//     PlcTask Inputs/GLOBAL.mtcs.parts.cover.parts.io.parts.slot11.wcState <-> WcState/WcState
//     PlcTask Outputs/GLOBAL.mtcs.parts.cover.parts.bottom.parts.p3.parts.motorRelay.digitalOutput <-> Channel 1/Output
//     PlcTask Outputs/GLOBAL.mtcs.parts.cover.parts.bottom.parts.p4.parts.motorRelay.digitalOutput <-> Channel 2/Output
//   MTCS/MTCS Instance <-> ECAT (EtherCAT)/Pumps room star point - coupler (EK1101)/Pumps room star point - Slot 1 (EK1122)/REM star point (CU1128)/Cover coupler (EK1101)/Cover slot 12 (relays magnet top-bot, EL2622)
//     PlcTask Inputs/GLOBAL.mtcs.parts.cover.parts.io.parts.slot12.infoData <-> InfoData/State
//     PlcTask Inputs/GLOBAL.mtcs.parts.cover.parts.io.parts.slot12.wcState <-> WcState/WcState
//     PlcTask Outputs/GLOBAL.mtcs.parts.cover.parts.bottom.parts.magnetsRelay.digitalOutput <-> Channel 2/Output
//     PlcTask Outputs/GLOBAL.mtcs.parts.cover.parts.top.parts.magnetsRelay.digitalOutput <-> Channel 1/Output
//   MTCS/MTCS Instance <-> ECAT (EtherCAT)/Pumps room star point - coupler (EK1101)/Pumps room star point - Slot 1 (EK1122)/REM star point (CU1128)/Cover coupler (EK1101)/Cover slot 13 (multimeter, EL3681)
//     PlcTask Inputs/GLOBAL.mtcs.parts.cover.currentMeasurement.error <-> SAI Inputs/Error
//     PlcTask Inputs/GLOBAL.mtcs.parts.cover.currentMeasurement.microAmpsValue <-> SAI Inputs/Value
//     PlcTask Inputs/GLOBAL.mtcs.parts.cover.parts.io.parts.slot13.infoData <-> InfoData/State
//     PlcTask Inputs/GLOBAL.mtcs.parts.cover.parts.io.parts.slot13.wcState <-> WcState/WcState
//   MTCS/MTCS Instance <-> ECAT (EtherCAT)/Pumps room star point - coupler (EK1101)/Pumps room star point - Slot 1 (EK1122)/REM star point (CU1128)/Cover coupler (EK1101)/Cover slot 2 (analog out, EL4008)
//     PlcTask Inputs/GLOBAL.mtcs.parts.cover.parts.io.parts.slot2.infoData <-> InfoData/State
//     PlcTask Inputs/GLOBAL.mtcs.parts.cover.parts.io.parts.slot2.wcState <-> WcState/WcState
//   MTCS/MTCS Instance <-> ECAT (EtherCAT)/Pumps room star point - coupler (EK1101)/Pumps room star point - Slot 1 (EK1122)/REM star point (CU1128)/Cover coupler (EK1101)/Cover slot 3 (digital in, EL1088)
//     PlcTask Inputs/GLOBAL.mtcs.parts.cover.parts.bottom.parts.p{1..4}.encoderErrorSignal <-> Channel {5..8}/Input  (4 links)
//     PlcTask Inputs/GLOBAL.mtcs.parts.cover.parts.io.parts.slot3.infoData <-> InfoData/State
//     PlcTask Inputs/GLOBAL.mtcs.parts.cover.parts.io.parts.slot3.wcState <-> WcState/WcState
//     PlcTask Inputs/GLOBAL.mtcs.parts.cover.parts.top.parts.p{1..4}.encoderErrorSignal <-> Channel {1..4}/Input  (4 links)
//   MTCS/MTCS Instance <-> ECAT (EtherCAT)/Pumps room star point - coupler (EK1101)/Pumps room star point - Slot 1 (EK1122)/REM star point (CU1128)/Cover coupler (EK1101)/Cover slot 4 (enc top 1-2, EL5002)
//     PlcTask Inputs/GLOBAL.mtcs.parts.cover.parts.io.parts.slot4.infoData <-> InfoData/State
//     PlcTask Inputs/GLOBAL.mtcs.parts.cover.parts.io.parts.slot4.wcState <-> WcState/WcState
//   MTCS/MTCS Instance <-> ECAT (EtherCAT)/Pumps room star point - coupler (EK1101)/Pumps room star point - Slot 1 (EK1122)/REM star point (CU1128)/Cover coupler (EK1101)/Cover slot 5 (enc top 3-4, EL5002)
//     PlcTask Inputs/GLOBAL.mtcs.parts.cover.parts.io.parts.slot5.infoData <-> InfoData/State
//     PlcTask Inputs/GLOBAL.mtcs.parts.cover.parts.io.parts.slot5.wcState <-> WcState/WcState
//   MTCS/MTCS Instance <-> ECAT (EtherCAT)/Pumps room star point - coupler (EK1101)/Pumps room star point - Slot 1 (EK1122)/REM star point (CU1128)/Cover coupler (EK1101)/Cover slot 6 (enc bot 1-2, EL5002)
//     PlcTask Inputs/GLOBAL.mtcs.parts.cover.parts.io.parts.slot6.infoData <-> InfoData/State
//     PlcTask Inputs/GLOBAL.mtcs.parts.cover.parts.io.parts.slot6.wcState <-> WcState/WcState
//   MTCS/MTCS Instance <-> ECAT (EtherCAT)/Pumps room star point - coupler (EK1101)/Pumps room star point - Slot 1 (EK1122)/REM star point (CU1128)/Cover coupler (EK1101)/Cover slot 7 (enc bot 3-4, EL5002)
//     PlcTask Inputs/GLOBAL.mtcs.parts.cover.parts.io.parts.slot7.infoData <-> InfoData/State
//     PlcTask Inputs/GLOBAL.mtcs.parts.cover.parts.io.parts.slot7.wcState <-> WcState/WcState
//   MTCS/MTCS Instance <-> ECAT (EtherCAT)/Pumps room star point - coupler (EK1101)/Pumps room star point - Slot 1 (EK1122)/REM star point (CU1128)/Cover coupler (EK1101)/Cover slot 8 (relays top 1-2, EL2622)
//     PlcTask Inputs/GLOBAL.mtcs.parts.cover.parts.io.parts.slot8.infoData <-> InfoData/State
//     PlcTask Inputs/GLOBAL.mtcs.parts.cover.parts.io.parts.slot8.wcState <-> WcState/WcState
//     PlcTask Outputs/GLOBAL.mtcs.parts.cover.parts.top.parts.p1.parts.motorRelay.digitalOutput <-> Channel 1/Output
//     PlcTask Outputs/GLOBAL.mtcs.parts.cover.parts.top.parts.p2.parts.motorRelay.digitalOutput <-> Channel 2/Output
//   MTCS/MTCS Instance <-> ECAT (EtherCAT)/Pumps room star point - coupler (EK1101)/Pumps room star point - Slot 1 (EK1122)/REM star point (CU1128)/Cover coupler (EK1101)/Cover slot 9 (relays top 3-4, EL2622)
//     PlcTask Inputs/GLOBAL.mtcs.parts.cover.parts.io.parts.slot9.infoData <-> InfoData/State
//     PlcTask Inputs/GLOBAL.mtcs.parts.cover.parts.io.parts.slot9.wcState <-> WcState/WcState
//     PlcTask Outputs/GLOBAL.mtcs.parts.cover.parts.top.parts.p3.parts.motorRelay.digitalOutput <-> Channel 1/Output
//     PlcTask Outputs/GLOBAL.mtcs.parts.cover.parts.top.parts.p4.parts.motorRelay.digitalOutput <-> Channel 2/Output
//   MTCS/MTCS Instance <-> ECAT (EtherCAT)/Pumps room star point - coupler (EK1101)/Pumps room star point - Slot 1 (EK1122)/REM star point (CU1128)/M1M2:COU (EK1101)
//     PlcTask Inputs/GLOBAL.mtcs.parts.m1.parts.io.parts.COU.infoData <-> InfoData/State
//     PlcTask Inputs/GLOBAL.mtcs.parts.m1.parts.io.parts.COU.wcState <-> WcState/WcState
//   MTCS/MTCS Instance <-> ECAT (EtherCAT)/Pumps room star point - coupler (EK1101)/Pumps room star point - Slot 1 (EK1122)/REM star point (CU1128)/M1M2:COU (EK1101)/M1M2:5V1 (Power 5V, EL9505)
//     PlcTask Inputs/GLOBAL.mtcs.parts.m1.parts.io.parts.P5V1.infoData <-> InfoData/State
//     PlcTask Inputs/GLOBAL.mtcs.parts.m1.parts.io.parts.P5V1.wcState <-> WcState/WcState
//   MTCS/MTCS Instance <-> ECAT (EtherCAT)/Pumps room star point - coupler (EK1101)/Pumps room star point - Slot 1 (EK1122)/REM star point (CU1128)/M1M2:COU (EK1101)/M1M2:AI1 (Analog in, EL3102)
//     PlcTask Inputs/GLOBAL.mtcs.parts.m1.parts.inclinometer.voltageMeasurement.error <-> AI Standard Channel 1/Status/Error
//     PlcTask Inputs/GLOBAL.mtcs.parts.m1.parts.inclinometer.voltageMeasurement.overrange <-> AI Standard Channel 1/Status/Overrange
//     PlcTask Inputs/GLOBAL.mtcs.parts.m1.parts.inclinometer.voltageMeasurement.rawValue <-> AI Standard Channel 1/Value
//     PlcTask Inputs/GLOBAL.mtcs.parts.m1.parts.inclinometer.voltageMeasurement.underrange <-> AI Standard Channel 1/Status/Underrange
//     PlcTask Inputs/GLOBAL.mtcs.parts.m1.parts.io.parts.AI1.infoData <-> InfoData/State
//     PlcTask Inputs/GLOBAL.mtcs.parts.m1.parts.io.parts.AI1.wcState <-> WcState/WcState
//   MTCS/MTCS Instance <-> ECAT (EtherCAT)/Pumps room star point - coupler (EK1101)/Pumps room star point - Slot 1 (EK1122)/REM star point (CU1128)/M1M2:COU (EK1101)/M1M2:AI2 (Analog in, EL3024)
//     PlcTask Inputs/GLOBAL.mtcs.parts.m1.parts.axialSupport.mirrorPressure.error <-> AI Standard Channel 2/Status/Error
//     PlcTask Inputs/GLOBAL.mtcs.parts.m1.parts.axialSupport.mirrorPressure.overrange <-> AI Standard Channel 2/Status/Overrange
//     PlcTask Inputs/GLOBAL.mtcs.parts.m1.parts.axialSupport.mirrorPressure.rawValue <-> AI Standard Channel 2/Value
//     PlcTask Inputs/GLOBAL.mtcs.parts.m1.parts.axialSupport.mirrorPressure.underrange <-> AI Standard Channel 2/Status/Underrange
//     PlcTask Inputs/GLOBAL.mtcs.parts.m1.parts.axialSupport.regulatorPressure.error <-> AI Standard Channel 1/Status/Error
//     PlcTask Inputs/GLOBAL.mtcs.parts.m1.parts.axialSupport.regulatorPressure.overrange <-> AI Standard Channel 1/Status/Overrange
//     PlcTask Inputs/GLOBAL.mtcs.parts.m1.parts.axialSupport.regulatorPressure.rawValue <-> AI Standard Channel 1/Value
//     PlcTask Inputs/GLOBAL.mtcs.parts.m1.parts.axialSupport.regulatorPressure.underrange <-> AI Standard Channel 1/Status/Underrange
//     PlcTask Inputs/GLOBAL.mtcs.parts.m1.parts.io.parts.AI2.infoData <-> InfoData/State
//     PlcTask Inputs/GLOBAL.mtcs.parts.m1.parts.io.parts.AI2.wcState <-> WcState/WcState
//     PlcTask Inputs/GLOBAL.mtcs.parts.m1.parts.radialSupport.mirrorPressure.error <-> AI Standard Channel 4/Status/Error
//     PlcTask Inputs/GLOBAL.mtcs.parts.m1.parts.radialSupport.mirrorPressure.overrange <-> AI Standard Channel 4/Status/Overrange
//     PlcTask Inputs/GLOBAL.mtcs.parts.m1.parts.radialSupport.mirrorPressure.rawValue <-> AI Standard Channel 4/Value
//     PlcTask Inputs/GLOBAL.mtcs.parts.m1.parts.radialSupport.mirrorPressure.underrange <-> AI Standard Channel 4/Status/Underrange
//     PlcTask Inputs/GLOBAL.mtcs.parts.m1.parts.radialSupport.regulatorPressure.error <-> AI Standard Channel 3/Status/Error
//     PlcTask Inputs/GLOBAL.mtcs.parts.m1.parts.radialSupport.regulatorPressure.overrange <-> AI Standard Channel 3/Status/Overrange
//     PlcTask Inputs/GLOBAL.mtcs.parts.m1.parts.radialSupport.regulatorPressure.rawValue <-> AI Standard Channel 3/Value
//     PlcTask Inputs/GLOBAL.mtcs.parts.m1.parts.radialSupport.regulatorPressure.underrange <-> AI Standard Channel 3/Status/Underrange
//   MTCS/MTCS Instance <-> ECAT (EtherCAT)/Pumps room star point - coupler (EK1101)/Pumps room star point - Slot 1 (EK1122)/REM star point (CU1128)/M1M2:COU (EK1101)/M1M2:AI3 (Analog in, EL3024)
//     PlcTask Inputs/GLOBAL.mtcs.parts.m1.parts.io.parts.AI3.infoData <-> InfoData/State
//     PlcTask Inputs/GLOBAL.mtcs.parts.m1.parts.io.parts.AI3.wcState <-> WcState/WcState
//     PlcTask Inputs/GLOBAL.mtcs.parts.m1.pneumaticSupplyPressure.error <-> AI Standard Channel 1/Status/Error
//     PlcTask Inputs/GLOBAL.mtcs.parts.m1.pneumaticSupplyPressure.overrange <-> AI Standard Channel 1/Status/Overrange
//     PlcTask Inputs/GLOBAL.mtcs.parts.m1.pneumaticSupplyPressure.rawValue <-> AI Standard Channel 1/Value
//     PlcTask Inputs/GLOBAL.mtcs.parts.m1.pneumaticSupplyPressure.underrange <-> AI Standard Channel 1/Status/Underrange
//   MTCS/MTCS Instance <-> ECAT (EtherCAT)/Pumps room star point - coupler (EK1101)/Pumps room star point - Slot 1 (EK1122)/REM star point (CU1128)/M1M2:COU (EK1101)/M1M2:AI4 (Analog in, EL3164)
//     PlcTask Inputs/GLOBAL.mtcs.parts.m1.parts.io.parts.AI4.infoData <-> InfoData/State
//     PlcTask Inputs/GLOBAL.mtcs.parts.m1.parts.io.parts.AI4.wcState <-> WcState/WcState
//     PlcTask Inputs/GLOBAL.mtcs.parts.m2.parts.tiltX.position.error <-> AI Standard Channel 1/Status/Error
//     PlcTask Inputs/GLOBAL.mtcs.parts.m2.parts.tiltX.position.overrange <-> AI Standard Channel 1/Status/Overrange
//     PlcTask Inputs/GLOBAL.mtcs.parts.m2.parts.tiltX.position.rawValue <-> AI Standard Channel 1/Value
//     PlcTask Inputs/GLOBAL.mtcs.parts.m2.parts.tiltX.position.underrange <-> AI Standard Channel 1/Status/Underrange
//     PlcTask Inputs/GLOBAL.mtcs.parts.m2.parts.tiltY.position.error <-> AI Standard Channel 3/Status/Error
//     PlcTask Inputs/GLOBAL.mtcs.parts.m2.parts.tiltY.position.overrange <-> AI Standard Channel 3/Status/Overrange
//     PlcTask Inputs/GLOBAL.mtcs.parts.m2.parts.tiltY.position.rawValue <-> AI Standard Channel 3/Value
//     PlcTask Inputs/GLOBAL.mtcs.parts.m2.parts.tiltY.position.underrange <-> AI Standard Channel 3/Status/Underrange
//     PlcTask Inputs/GLOBAL.mtcs.parts.m2.parts.x.position.error <-> AI Standard Channel 2/Status/Error
//     PlcTask Inputs/GLOBAL.mtcs.parts.m2.parts.x.position.overrange <-> AI Standard Channel 2/Status/Overrange
//     PlcTask Inputs/GLOBAL.mtcs.parts.m2.parts.x.position.rawValue <-> AI Standard Channel 2/Value
//     PlcTask Inputs/GLOBAL.mtcs.parts.m2.parts.x.position.underrange <-> AI Standard Channel 2/Status/Underrange
//     PlcTask Inputs/GLOBAL.mtcs.parts.m2.parts.y.position.error <-> AI Standard Channel 4/Status/Error
//     PlcTask Inputs/GLOBAL.mtcs.parts.m2.parts.y.position.overrange <-> AI Standard Channel 4/Status/Overrange
//     PlcTask Inputs/GLOBAL.mtcs.parts.m2.parts.y.position.rawValue <-> AI Standard Channel 4/Value
//     PlcTask Inputs/GLOBAL.mtcs.parts.m2.parts.y.position.underrange <-> AI Standard Channel 4/Status/Underrange
//   MTCS/MTCS Instance <-> ECAT (EtherCAT)/Pumps room star point - coupler (EK1101)/Pumps room star point - Slot 1 (EK1122)/REM star point (CU1128)/M1M2:COU (EK1101)/M1M2:AO1 (Analog out, EL4022)
//     PlcTask Inputs/GLOBAL.mtcs.parts.m1.parts.io.parts.AO1.infoData <-> InfoData/State
//     PlcTask Inputs/GLOBAL.mtcs.parts.m1.parts.io.parts.AO1.wcState <-> WcState/WcState
//     PlcTask Outputs/GLOBAL.mtcs.parts.m1.parts.axialSupport.pressureSetpointOutput <-> AO Outputs Channel 1/Analog output
//     PlcTask Outputs/GLOBAL.mtcs.parts.m1.parts.radialSupport.pressureSetpointOutput <-> AO Outputs Channel 2/Analog output
//   MTCS/MTCS Instance <-> ECAT (EtherCAT)/Pumps room star point - coupler (EK1101)/Pumps room star point - Slot 1 (EK1122)/REM star point (CU1128)/M1M2:COU (EK1101)/M1M2:DO1 (Digital out, EL2024)
//     PlcTask Inputs/GLOBAL.mtcs.parts.m1.parts.io.parts.DO1.infoData <-> InfoData/State
//     PlcTask Inputs/GLOBAL.mtcs.parts.m1.parts.io.parts.DO1.wcState <-> WcState/WcState
//     PlcTask Outputs/GLOBAL.mtcs.parts.m1.parts.radialSupport.parts.vacuumRelay.digitalOutput <-> Channel 1/Output
//     PlcTask Outputs/GLOBAL.mtcs.parts.m2.parts.heater.digitalOutput <-> Channel 2/Output
//   MTCS/MTCS Instance <-> ECAT (EtherCAT)/Pumps room star point - coupler (EK1101)/Pumps room star point - Slot 1 (EK1122)/REM star point (CU1128)/M1M2:COU (EK1101)/M1M2:DO2 (Digital out, EL2124)
//     PlcTask Inputs/GLOBAL.mtcs.parts.m1.parts.io.parts.DO2.infoData <-> InfoData/State
//     PlcTask Inputs/GLOBAL.mtcs.parts.m1.parts.io.parts.DO2.wcState <-> WcState/WcState
//     PlcTask Outputs/GLOBAL.mtcs.parts.m2.parts.multiplexer.parts.A.digitalOutput <-> Channel 3/Output
//     PlcTask Outputs/GLOBAL.mtcs.parts.m2.parts.multiplexer.parts.B.digitalOutput <-> Channel 2/Output
//     PlcTask Outputs/GLOBAL.mtcs.parts.m2.parts.multiplexer.parts.C.digitalOutput <-> Channel 4/Output
//     PlcTask Outputs/GLOBAL.mtcs.parts.m2.parts.multiplexer.parts.driveEnable.digitalOutput <-> Channel 1/Output
//   MTCS/MTCS Instance <-> ECAT (EtherCAT)/Pumps room star point - coupler (EK1101)/Pumps room star point - Slot 1 (EK1122)/REM star point (CU1128)/M1M2:COU (EK1101)/M1M2:DO3 (Digital out, EL2124)
//     PlcFastTask Outputs/GLOBAL.mtcs.parts.m2.parts.multiplexer.parts.release.digitalOutput <-> Channel 3/Output
//     PlcTask Inputs/GLOBAL.mtcs.parts.m1.parts.io.parts.DO3.infoData <-> InfoData/State
//     PlcTask Inputs/GLOBAL.mtcs.parts.m1.parts.io.parts.DO3.wcState <-> WcState/WcState
//     PlcTask Outputs/GLOBAL.mtcs.parts.m2.parts.multiplexer.parts.CW.digitalOutput <-> Channel 1/Output
//     PlcTask Outputs/GLOBAL.mtcs.parts.m2.parts.z.parts.highSpeed.digitalOutput <-> Channel 2/Output
//   MTCS/MTCS Instance <-> ECAT (EtherCAT)/Pumps room star point - coupler (EK1101)/Pumps room star point - Slot 1 (EK1122)/REM star point (CU1128)/M1M2:COU (EK1101)/M1M2:INC1 (Counter, EL5101)
//     PlcFastTask Inputs/FAST.m2FastTaskControl.setCounterDone <-> ENC Status/Status/Set counter done
//     PlcFastTask Inputs/GLOBAL.mtcs.parts.m2.parts.moveStepsProcedure.actualCounterValue <-> ENC Status/Counter value
//     PlcFastTask Outputs/FAST.m2FastTaskControl.setCounter <-> ENC Control/Control/Set counter
//     PlcFastTask Outputs/FAST.m2FastTaskControl.setCounterValue <-> ENC Control/Set counter value
//     PlcTask Inputs/GLOBAL.mtcs.parts.m1.parts.io.parts.INC1.infoData <-> InfoData/State
//     PlcTask Inputs/GLOBAL.mtcs.parts.m1.parts.io.parts.INC1.wcState <-> WcState/WcState
//     PlcTask Inputs/GLOBAL.mtcs.parts.m2.parts.multiplexer.noFault <-> ENC Status/Status/Status of input status
//   MTCS/MTCS Instance <-> ECAT (EtherCAT)/Pumps room star point - coupler (EK1101)/Pumps room star point - Slot 1 (EK1122)/REM star point (CU1128)/M1M2:COU (EK1101)/M1M2:PWR1 (Power supply, EL9410)
//     PlcTask Inputs/GLOBAL.mtcs.parts.m1.parts.io.parts.PWR1.infoData <-> InfoData/State
//     PlcTask Inputs/GLOBAL.mtcs.parts.m1.parts.io.parts.PWR1.wcState <-> WcState/WcState
//   MTCS/MTCS Instance <-> ECAT (EtherCAT)/Pumps room star point - coupler (EK1101)/Pumps room star point - Slot 1 (EK1122)/REM star point (CU1128)/M1M2:COU (EK1101)/M1M2:RE1 (Relay, EL2622)
//     PlcTask Inputs/GLOBAL.mtcs.parts.m1.parts.io.parts.RE1.infoData <-> InfoData/State
//     PlcTask Inputs/GLOBAL.mtcs.parts.m1.parts.io.parts.RE1.wcState <-> WcState/WcState
//     PlcTask Outputs/GLOBAL.mtcs.parts.m2.parts.powerRelay.digitalOutput <-> Channel 1/Output
//   MTCS/MTCS Instance <-> ECAT (EtherCAT)/Pumps room star point - coupler (EK1101)/Pumps room star point - Slot 1 (EK1122)/REM star point (CU1128)/M1M2:COU (EK1101)/M1M2:RES1 (Res bridge SO, EL3351)
//     PlcTask Inputs/GLOBAL.mtcs.parts.m1.parts.axialSupport.mirrorSouthForce.error <-> AIBridge Inputs/Error
//     PlcTask Inputs/GLOBAL.mtcs.parts.m1.parts.axialSupport.mirrorSouthForce.overrange <-> AIBridge Inputs/Overrange
//     PlcTask Inputs/GLOBAL.mtcs.parts.m1.parts.axialSupport.mirrorSouthForce.rawValue <-> AIBridge Inputs/Value
//     PlcTask Inputs/GLOBAL.mtcs.parts.m1.parts.axialSupport.mirrorSouthForce.underrange <-> AIBridge Inputs/Underrange
//     PlcTask Inputs/GLOBAL.mtcs.parts.m1.parts.io.parts.RES1.infoData <-> InfoData/State
//     PlcTask Inputs/GLOBAL.mtcs.parts.m1.parts.io.parts.RES1.wcState <-> WcState/WcState
//   MTCS/MTCS Instance <-> ECAT (EtherCAT)/Pumps room star point - coupler (EK1101)/Pumps room star point - Slot 1 (EK1122)/REM star point (CU1128)/M1M2:COU (EK1101)/M1M2:RES2 (Res bridge NE, EL3351)
//     PlcTask Inputs/GLOBAL.mtcs.parts.m1.parts.axialSupport.mirrorNorthEastForce.error <-> AIBridge Inputs/Error
//     PlcTask Inputs/GLOBAL.mtcs.parts.m1.parts.axialSupport.mirrorNorthEastForce.overrange <-> AIBridge Inputs/Overrange
//     PlcTask Inputs/GLOBAL.mtcs.parts.m1.parts.axialSupport.mirrorNorthEastForce.rawValue <-> AIBridge Inputs/Value
//     PlcTask Inputs/GLOBAL.mtcs.parts.m1.parts.axialSupport.mirrorNorthEastForce.underrange <-> AIBridge Inputs/Underrange
//     PlcTask Inputs/GLOBAL.mtcs.parts.m1.parts.io.parts.RES2.infoData <-> InfoData/State
//     PlcTask Inputs/GLOBAL.mtcs.parts.m1.parts.io.parts.RES2.wcState <-> WcState/WcState
//   MTCS/MTCS Instance <-> ECAT (EtherCAT)/Pumps room star point - coupler (EK1101)/Pumps room star point - Slot 1 (EK1122)/REM star point (CU1128)/M1M2:COU (EK1101)/M1M2:RES3 (Res bridge NW, EL3351)
//     PlcTask Inputs/GLOBAL.mtcs.parts.m1.parts.axialSupport.mirrorNorthWestForce.error <-> AIBridge Inputs/Error
//     PlcTask Inputs/GLOBAL.mtcs.parts.m1.parts.axialSupport.mirrorNorthWestForce.overrange <-> AIBridge Inputs/Overrange
//     PlcTask Inputs/GLOBAL.mtcs.parts.m1.parts.axialSupport.mirrorNorthWestForce.rawValue <-> AIBridge Inputs/Value
//     PlcTask Inputs/GLOBAL.mtcs.parts.m1.parts.axialSupport.mirrorNorthWestForce.underrange <-> AIBridge Inputs/Underrange
//     PlcTask Inputs/GLOBAL.mtcs.parts.m1.parts.io.parts.RES3.infoData <-> InfoData/State
//     PlcTask Inputs/GLOBAL.mtcs.parts.m1.parts.io.parts.RES3.wcState <-> WcState/WcState
//   MTCS/MTCS Instance <-> ECAT (EtherCAT)/Pumps room star point - coupler (EK1101)/Pumps room star point - Slot 1 (EK1122)/REM star point (CU1128)/M1M2:COU (EK1101)/M1M2:SSI1 (SSI encoder, EL5001)
//     PlcTask Inputs/GLOBAL.mtcs.parts.m1.parts.io.parts.SSI1.infoData <-> InfoData/State
//     PlcTask Inputs/GLOBAL.mtcs.parts.m1.parts.io.parts.SSI1.wcState <-> WcState/WcState
//     PlcTask Inputs/GLOBAL.mtcs.parts.m2.parts.z.parts.encoder.counterValue <-> SSI Inputs/Counter value
//     PlcTask Inputs/GLOBAL.mtcs.parts.m2.parts.z.parts.encoder.dataError <-> SSI Inputs/Status/Data error
//     PlcTask Inputs/GLOBAL.mtcs.parts.m2.parts.z.parts.encoder.frameError <-> SSI Inputs/Status/Frame error
//     PlcTask Inputs/GLOBAL.mtcs.parts.m2.parts.z.parts.encoder.powerFailure <-> SSI Inputs/Status/Power failure
//     PlcTask Inputs/GLOBAL.mtcs.parts.m2.parts.z.parts.encoder.syncError <-> SSI Inputs/Status/Sync error
//   MTCS/MTCS Instance <-> ECAT (EtherCAT)/Pumps room star point - coupler (EK1101)/Pumps room star point - Slot 1 (EK1122)/REM star point (CU1128)/REM star point B (CU1128-B)/Accelerometer box (EP1816-3008)
//     PlcTask Inputs/GLOBAL.mtcs.parts.telemetry.parts.accelerometers.tube.X1plus.error <-> AI Inputs Channel 1/Status/Error
//     PlcTask Inputs/GLOBAL.mtcs.parts.telemetry.parts.accelerometers.tube.X1plus.milliGValue <-> AI Inputs Channel 1/Value
//     PlcTask Inputs/GLOBAL.mtcs.parts.telemetry.parts.accelerometers.tube.X2minus.error <-> AI Inputs Channel 5/Status/Error
//     PlcTask Inputs/GLOBAL.mtcs.parts.telemetry.parts.accelerometers.tube.X2minus.milliGValue <-> AI Inputs Channel 5/Value
//     PlcTask Inputs/GLOBAL.mtcs.parts.telemetry.parts.accelerometers.tube.Y1plus.error <-> AI Inputs Channel 2/Status/Error
//     PlcTask Inputs/GLOBAL.mtcs.parts.telemetry.parts.accelerometers.tube.Y2plus.error <-> AI Inputs Channel 4/Status/Error
//     PlcTask Inputs/GLOBAL.mtcs.parts.telemetry.parts.accelerometers.tube.Y1plus.milliGValue <-> AI Inputs Channel 2/Value
//     PlcTask Inputs/GLOBAL.mtcs.parts.telemetry.parts.accelerometers.tube.Y2plus.milliGValue <-> AI Inputs Channel 4/Value
//     PlcTask Inputs/GLOBAL.mtcs.parts.telemetry.parts.accelerometers.tube.Z1minus.error <-> AI Inputs Channel 3/Status/Error
//     PlcTask Inputs/GLOBAL.mtcs.parts.telemetry.parts.accelerometers.tube.Z2minus.error <-> AI Inputs Channel 6/Status/Error
//     PlcTask Inputs/GLOBAL.mtcs.parts.telemetry.parts.accelerometers.tube.Z1minus.milliGValue <-> AI Inputs Channel 3/Value
//     PlcTask Inputs/GLOBAL.mtcs.parts.telemetry.parts.accelerometers.tube.Z2minus.milliGValue <-> AI Inputs Channel 6/Value
//     PlcTask Inputs/GLOBAL.mtcs.parts.telemetry.parts.io.parts.tubeAccelerometers.infoData <-> InfoData/State
//     PlcTask Inputs/GLOBAL.mtcs.parts.telemetry.parts.io.parts.tubeAccelerometers.wcState <-> WcState/WcState
//   MTCS/MTCS Instance <-> ECAT (EtherCAT)/Pumps room star point - coupler (EK1101)/Pumps room star point - Slot 1 (EK1122)/REM star point (CU1128)/REM star point B (CU1128-B)/M3 coupler (EK1100)
//     PlcTask Inputs/GLOBAL.mtcs.parts.m3.parts.io.parts.coupler.infoData <-> InfoData/State
//   MTCS/MTCS Instance <-> ECAT (EtherCAT)/Pumps room star point - coupler (EK1101)/Pumps room star point - Slot 1 (EK1122)/REM star point (CU1128)/REM star point B (CU1128-B)/M3 coupler (EK1100)/M3 Slot 1 (digital in EL1088)
//     PlcTask Inputs/GLOBAL.mtcs.parts.m3.parts.io.parts.slot1.infoData <-> InfoData/State
//     PlcTask Inputs/GLOBAL.mtcs.parts.m3.parts.io.parts.slot1.wcState <-> WcState/WcState
//     PlcTask Inputs/GLOBAL.mtcs.parts.m3.parts.rotation.negativeLimitSwitchActive <-> Channel 4/ROT limit switch -
//     PlcTask Inputs/GLOBAL.mtcs.parts.m3.parts.rotation.positiveLimitSwitchActive <-> Channel 2/ROT limit switch +
//     PlcTask Inputs/GLOBAL.mtcs.parts.m3.parts.translation.negativeLimitSwitchActive <-> Channel 3/LIN limit switch -
//     PlcTask Inputs/GLOBAL.mtcs.parts.m3.parts.translation.positiveLimitSwitchActive <-> Channel 1/LIN limit switch +
//   MTCS/MTCS Instance <-> ECAT (EtherCAT)/Pumps room star point - coupler (EK1101)/Pumps room star point - Slot 1 (EK1122)/REM star point (CU1128)/REM star point B (CU1128-B)/M3 coupler (EK1100)/M3 Slot 2 (encoder EL5101)
//     PlcTask Inputs/GLOBAL.mtcs.parts.m3.parts.io.parts.slot2.infoData <-> InfoData/State
//     PlcTask Inputs/GLOBAL.mtcs.parts.m3.parts.io.parts.slot2.wcState <-> WcState/WcState
//   MTCS/MTCS Instance <-> ECAT (EtherCAT)/Pumps room star point - coupler (EK1101)/Pumps room star point - Slot 1 (EK1122)/REM star point (CU1128)/REM star point B (CU1128-B)/M3 coupler (EK1100)/M3 Slot 3 (encoder EL5001)
//     PlcTask Inputs/GLOBAL.mtcs.parts.m3.parts.io.parts.slot3.infoData <-> InfoData/State
//     PlcTask Inputs/GLOBAL.mtcs.parts.m3.parts.io.parts.slot3.wcState <-> WcState/WcState
//   MTCS/MTCS Instance <-> ECAT (EtherCAT)/Pumps room star point - coupler (EK1101)/Pumps room star point - Slot 1 (EK1122)/REM star point (CU1128)/REM star point B (CU1128-B)/M3 coupler (EK1100)/M3 Slot 4 (CANopen EL6751)
//     PlcTask Inputs/GLOBAL.mtcs.parts.m3.parts.io.parts.slot4.infoData <-> InfoData/State
//   MTCS/MTCS Instance <-> ECAT (EtherCAT)/Pumps room star point - coupler (EK1101)/Pumps room star point - Slot 1 (EK1122)/REM star point (CU1128)/REM star point B (CU1128-B)/Telemetry coupler (EK1101)
//     PlcTask Inputs/GLOBAL.mtcs.parts.telemetry.parts.io.parts.coupler.infoData <-> InfoData/State
//     PlcTask Inputs/GLOBAL.mtcs.parts.telemetry.parts.io.parts.coupler.wcState <-> WcState/WcState
//   MTCS/MTCS Instance <-> ECAT (EtherCAT)/Pumps room star point - coupler (EK1101)/Pumps room star point - Slot 1 (EK1122)/REM star point (CU1128)/REM star point B (CU1128-B)/Telemetry coupler (EK1101)/Slot 10 (EL3202-0010)
//     PlcTask Inputs/GLOBAL.mtcs.parts.telemetry.parts.io.parts.slot10.infoData <-> InfoData/State
//     PlcTask Inputs/GLOBAL.mtcs.parts.telemetry.parts.io.parts.slot10.wcState <-> WcState/WcState
//     PlcTask Inputs/GLOBAL.mtcs.parts.telemetry.parts.temperatures.hermesTelescopeAdapter.error <-> RTD Inputs Channel 1/Status/Error
//     PlcTask Inputs/GLOBAL.mtcs.parts.telemetry.parts.temperatures.hermesTelescopeAdapter.overrange <-> RTD Inputs Channel 1/Status/Overrange
//     PlcTask Inputs/GLOBAL.mtcs.parts.telemetry.parts.temperatures.hermesTelescopeAdapter.rawValue <-> RTD Inputs Channel 1/Value
//     PlcTask Inputs/GLOBAL.mtcs.parts.telemetry.parts.temperatures.hermesTelescopeAdapter.underrange <-> RTD Inputs Channel 1/Status/Underrange
//   MTCS/MTCS Instance <-> ECAT (EtherCAT)/Pumps room star point - coupler (EK1101)/Pumps room star point - Slot 1 (EK1122)/REM star point (CU1128)/REM star point B (CU1128-B)/Telemetry coupler (EK1101)/Slot 11 (EL3202-0010)
//     PlcTask Inputs/GLOBAL.mtcs.parts.telemetry.parts.io.parts.slot11.infoData <-> InfoData/State
//     PlcTask Inputs/GLOBAL.mtcs.parts.telemetry.parts.io.parts.slot11.wcState <-> WcState/WcState
//     PlcTask Inputs/GLOBAL.mtcs.parts.telemetry.parts.temperatures.insideTube.error <-> RTD Inputs Channel 2/Status/Error
//     PlcTask Inputs/GLOBAL.mtcs.parts.telemetry.parts.temperatures.insideTube.overrange <-> RTD Inputs Channel 2/Status/Overrange
//     PlcTask Inputs/GLOBAL.mtcs.parts.telemetry.parts.temperatures.insideTube.rawValue <-> RTD Inputs Channel 2/Value
//     PlcTask Inputs/GLOBAL.mtcs.parts.telemetry.parts.temperatures.insideTube.underrange <-> RTD Inputs Channel 2/Status/Underrange
//     PlcTask Inputs/GLOBAL.mtcs.parts.telemetry.parts.temperatures.topAir.error <-> RTD Inputs Channel 1/Status/Error
//     PlcTask Inputs/GLOBAL.mtcs.parts.telemetry.parts.temperatures.topAir.overrange <-> RTD Inputs Channel 1/Status/Overrange
//     PlcTask Inputs/GLOBAL.mtcs.parts.telemetry.parts.temperatures.topAir.rawValue <-> RTD Inputs Channel 1/Value
//     PlcTask Inputs/GLOBAL.mtcs.parts.telemetry.parts.temperatures.topAir.underrange <-> RTD Inputs Channel 1/Status/Underrange
//   MTCS/MTCS Instance <-> ECAT (EtherCAT)/Pumps room star point - coupler (EK1101)/Pumps room star point - Slot 1 (EK1122)/REM star point (CU1128)/REM star point B (CU1128-B)/Telemetry coupler (EK1101)/Slot 12 (EL3024)
//     PlcTask Inputs/GLOBAL.mtcs.parts.telemetry.parts.io.parts.slot12.infoData <-> InfoData/State
//     PlcTask Inputs/GLOBAL.mtcs.parts.telemetry.parts.io.parts.slot12.wcState <-> WcState/WcState
//     PlcTask Inputs/GLOBAL.mtcs.parts.telemetry.parts.relativeHumidities.insideTube.error <-> AI Standard Channel 3/Status/Error
//     PlcTask Inputs/GLOBAL.mtcs.parts.telemetry.parts.relativeHumidities.insideTube.overrange <-> AI Standard Channel 3/Status/Overrange
//     PlcTask Inputs/GLOBAL.mtcs.parts.telemetry.parts.relativeHumidities.insideTube.rawValue <-> AI Standard Channel 3/Value
//     PlcTask Inputs/GLOBAL.mtcs.parts.telemetry.parts.relativeHumidities.insideTube.underrange <-> AI Standard Channel 3/Status/Underrange
//     PlcTask Inputs/GLOBAL.mtcs.parts.telemetry.parts.relativeHumidities.topAir.error <-> AI Standard Channel 1/Status/Error
//     PlcTask Inputs/GLOBAL.mtcs.parts.telemetry.parts.relativeHumidities.topAir.overrange <-> AI Standard Channel 1/Status/Overrange
//     PlcTask Inputs/GLOBAL.mtcs.parts.telemetry.parts.relativeHumidities.topAir.rawValue <-> AI Standard Channel 1/Value
//     PlcTask Inputs/GLOBAL.mtcs.parts.telemetry.parts.relativeHumidities.topAir.underrange <-> AI Standard Channel 1/Status/Underrange
//   MTCS/MTCS Instance <-> ECAT (EtherCAT)/Pumps room star point - coupler (EK1101)/Pumps room star point - Slot 1 (EK1122)/REM star point (CU1128)/REM star point B (CU1128-B)/Telemetry coupler (EK1101)/Slot 13 (EL2008)
//     PlcTask Inputs/GLOBAL.mtcs.parts.telemetry.parts.io.parts.slot13.infoData <-> InfoData/State
//     PlcTask Inputs/GLOBAL.mtcs.parts.telemetry.parts.io.parts.slot13.wcState <-> WcState/WcState
//     PlcTask Outputs/GLOBAL.mtcs.parts.telemetry.parts.flatfieldLeds.parts.output{1..8}.digitalOutput <-> Channel {1..8}/Output  (8 links)
//   MTCS/MTCS Instance <-> ECAT (EtherCAT)/Pumps room star point - coupler (EK1101)/Pumps room star point - Slot 1 (EK1122)/REM star point (CU1128)/REM star point B (CU1128-B)/Telemetry coupler (EK1101)/Slot 5 (EL3202-0010)
//     PlcTask Inputs/GLOBAL.mtcs.parts.telemetry.parts.io.parts.slot5.infoData <-> InfoData/State
//     PlcTask Inputs/GLOBAL.mtcs.parts.telemetry.parts.io.parts.slot5.wcState <-> WcState/WcState
//     PlcTask Inputs/GLOBAL.mtcs.parts.telemetry.parts.temperatures.m1.error <-> RTD Inputs Channel 1/Status/Error
//     PlcTask Inputs/GLOBAL.mtcs.parts.telemetry.parts.temperatures.m1.overrange <-> RTD Inputs Channel 1/Status/Overrange
//     PlcTask Inputs/GLOBAL.mtcs.parts.telemetry.parts.temperatures.m1.rawValue <-> RTD Inputs Channel 1/Value
//     PlcTask Inputs/GLOBAL.mtcs.parts.telemetry.parts.temperatures.m1.underrange <-> RTD Inputs Channel 1/Status/Underrange
//     PlcTask Inputs/GLOBAL.mtcs.parts.telemetry.parts.temperatures.mirrorCell.error <-> RTD Inputs Channel 2/Status/Error
//     PlcTask Inputs/GLOBAL.mtcs.parts.telemetry.parts.temperatures.mirrorCell.overrange <-> RTD Inputs Channel 2/Status/Overrange
//     PlcTask Inputs/GLOBAL.mtcs.parts.telemetry.parts.temperatures.mirrorCell.rawValue <-> RTD Inputs Channel 2/Value
//     PlcTask Inputs/GLOBAL.mtcs.parts.telemetry.parts.temperatures.mirrorCell.underrange <-> RTD Inputs Channel 2/Status/Underrange
//   MTCS/MTCS Instance <-> ECAT (EtherCAT)/Pumps room star point - coupler (EK1101)/Pumps room star point - Slot 1 (EK1122)/REM star point (CU1128)/REM star point B (CU1128-B)/Telemetry coupler (EK1101)/Slot 6 (EL3202-0010)
//     PlcTask Inputs/GLOBAL.mtcs.parts.telemetry.parts.io.parts.slot6.infoData <-> InfoData/State
//     PlcTask Inputs/GLOBAL.mtcs.parts.telemetry.parts.io.parts.slot6.wcState <-> WcState/WcState
//     PlcTask Inputs/GLOBAL.mtcs.parts.telemetry.parts.temperatures.m2.error <-> RTD Inputs Channel 1/Status/Error
//     PlcTask Inputs/GLOBAL.mtcs.parts.telemetry.parts.temperatures.m2.overrange <-> RTD Inputs Channel 1/Status/Overrange
//     PlcTask Inputs/GLOBAL.mtcs.parts.telemetry.parts.temperatures.m2.rawValue <-> RTD Inputs Channel 1/Value
//     PlcTask Inputs/GLOBAL.mtcs.parts.telemetry.parts.temperatures.m2.underrange <-> RTD Inputs Channel 1/Status/Underrange
//     PlcTask Inputs/GLOBAL.mtcs.parts.telemetry.parts.temperatures.m2Electronics.error <-> RTD Inputs Channel 2/Status/Error
//     PlcTask Inputs/GLOBAL.mtcs.parts.telemetry.parts.temperatures.m2Electronics.overrange <-> RTD Inputs Channel 2/Status/Overrange
//     PlcTask Inputs/GLOBAL.mtcs.parts.telemetry.parts.temperatures.m2Electronics.rawValue <-> RTD Inputs Channel 2/Value
//     PlcTask Inputs/GLOBAL.mtcs.parts.telemetry.parts.temperatures.m2Electronics.underrange <-> RTD Inputs Channel 2/Status/Underrange
//   MTCS/MTCS Instance <-> ECAT (EtherCAT)/Pumps room star point - coupler (EK1101)/Pumps room star point - Slot 1 (EK1122)/REM star point (CU1128)/REM star point B (CU1128-B)/Telemetry coupler (EK1101)/Slot 7 (EL3202-0010)
//     PlcTask Inputs/GLOBAL.mtcs.parts.telemetry.parts.io.parts.slot7.infoData <-> InfoData/State
//     PlcTask Inputs/GLOBAL.mtcs.parts.telemetry.parts.io.parts.slot7.wcState <-> WcState/WcState
//     PlcTask Inputs/GLOBAL.mtcs.parts.telemetry.parts.temperatures.centreTube.error <-> RTD Inputs Channel 2/Status/Error
//     PlcTask Inputs/GLOBAL.mtcs.parts.telemetry.parts.temperatures.centreTube.overrange <-> RTD Inputs Channel 2/Status/Overrange
//     PlcTask Inputs/GLOBAL.mtcs.parts.telemetry.parts.temperatures.centreTube.rawValue <-> RTD Inputs Channel 2/Value
//     PlcTask Inputs/GLOBAL.mtcs.parts.telemetry.parts.temperatures.centreTube.underrange <-> RTD Inputs Channel 2/Status/Underrange
//     PlcTask Inputs/GLOBAL.mtcs.parts.telemetry.parts.temperatures.topTube.error <-> RTD Inputs Channel 1/Status/Error
//     PlcTask Inputs/GLOBAL.mtcs.parts.telemetry.parts.temperatures.topTube.overrange <-> RTD Inputs Channel 1/Status/Overrange
//     PlcTask Inputs/GLOBAL.mtcs.parts.telemetry.parts.temperatures.topTube.rawValue <-> RTD Inputs Channel 1/Value
//     PlcTask Inputs/GLOBAL.mtcs.parts.telemetry.parts.temperatures.topTube.underrange <-> RTD Inputs Channel 1/Status/Underrange
//   MTCS/MTCS Instance <-> ECAT (EtherCAT)/Pumps room star point - coupler (EK1101)/Pumps room star point - Slot 1 (EK1122)/REM star point (CU1128)/REM star point B (CU1128-B)/Telemetry coupler (EK1101)/Slot 8 (EL3202-0010)
//     PlcTask Inputs/GLOBAL.mtcs.parts.telemetry.parts.io.parts.slot8.infoData <-> InfoData/State
//     PlcTask Inputs/GLOBAL.mtcs.parts.telemetry.parts.io.parts.slot8.wcState <-> WcState/WcState
//     PlcTask Inputs/GLOBAL.mtcs.parts.telemetry.parts.temperatures.fork.error <-> RTD Inputs Channel 1/Status/Error
//     PlcTask Inputs/GLOBAL.mtcs.parts.telemetry.parts.temperatures.fork.overrange <-> RTD Inputs Channel 1/Status/Overrange
//     PlcTask Inputs/GLOBAL.mtcs.parts.telemetry.parts.temperatures.fork.rawValue <-> RTD Inputs Channel 1/Value
//     PlcTask Inputs/GLOBAL.mtcs.parts.telemetry.parts.temperatures.fork.underrange <-> RTD Inputs Channel 1/Status/Underrange
//     PlcTask Inputs/GLOBAL.mtcs.parts.telemetry.parts.temperatures.nasmythAir.error <-> RTD Inputs Channel 2/Status/Error
//     PlcTask Inputs/GLOBAL.mtcs.parts.telemetry.parts.temperatures.nasmythAir.overrange <-> RTD Inputs Channel 2/Status/Overrange
//     PlcTask Inputs/GLOBAL.mtcs.parts.telemetry.parts.temperatures.nasmythAir.rawValue <-> RTD Inputs Channel 2/Value
//     PlcTask Inputs/GLOBAL.mtcs.parts.telemetry.parts.temperatures.nasmythAir.underrange <-> RTD Inputs Channel 2/Status/Underrange
//   MTCS/MTCS Instance <-> ECAT (EtherCAT)/Pumps room star point - coupler (EK1101)/Pumps room star point - Slot 1 (EK1122)/REM star point (CU1128)/REM star point B (CU1128-B)/Telemetry coupler (EK1101)/Slot 9 (EL3202-0010)
//     PlcTask Inputs/GLOBAL.mtcs.parts.telemetry.parts.io.parts.slot9.infoData <-> InfoData/State
//     PlcTask Inputs/GLOBAL.mtcs.parts.telemetry.parts.io.parts.slot9.wcState <-> WcState/WcState
//     PlcTask Inputs/GLOBAL.mtcs.parts.telemetry.parts.temperatures.rem.error <-> RTD Inputs Channel 1/Status/Error
//     PlcTask Inputs/GLOBAL.mtcs.parts.telemetry.parts.temperatures.rem.overrange <-> RTD Inputs Channel 1/Status/Overrange
//     PlcTask Inputs/GLOBAL.mtcs.parts.telemetry.parts.temperatures.rem.rawValue <-> RTD Inputs Channel 1/Value
//     PlcTask Inputs/GLOBAL.mtcs.parts.telemetry.parts.temperatures.rem.underrange <-> RTD Inputs Channel 1/Status/Underrange
//     PlcTask Inputs/GLOBAL.mtcs.parts.telemetry.parts.temperatures.rpm.error <-> RTD Inputs Channel 2/Status/Error
//     PlcTask Inputs/GLOBAL.mtcs.parts.telemetry.parts.temperatures.rpm.overrange <-> RTD Inputs Channel 2/Status/Overrange
//     PlcTask Inputs/GLOBAL.mtcs.parts.telemetry.parts.temperatures.rpm.rawValue <-> RTD Inputs Channel 2/Value
//     PlcTask Inputs/GLOBAL.mtcs.parts.telemetry.parts.temperatures.rpm.underrange <-> RTD Inputs Channel 2/Status/Underrange
//   MTCS/MTCS Instance <-> ECAT (EtherCAT)/Pumps room star point - coupler (EK1101)/Pumps room star point - Slot 1 (EK1122)/REM star point (CU1128)/REM star point C (CU1128-C)/ABLD (AX5206-0000-0203)
//     PlcFastTask Inputs/GLOBAL.mtcs.parts.axes.parts.io.parts.ablDrive.parts.channelA.digitalInputs <-> AT 1/Digital inputs, state
//     PlcFastTask Inputs/GLOBAL.mtcs.parts.axes.parts.io.parts.ablDrive.parts.channelA.errorC1D <-> AT 1/Class 1 diagnostic (C1D)
//     PlcFastTask Inputs/GLOBAL.mtcs.parts.axes.parts.io.parts.ablDrive.parts.channelA.safetyOptionState <-> AT 1/Safety option state
//     PlcFastTask Inputs/GLOBAL.mtcs.parts.axes.parts.io.parts.ablDrive.parts.channelA.torqueFeedbackValue <-> AT 1/Torque feedback value
//     PlcFastTask Inputs/GLOBAL.mtcs.parts.axes.parts.io.parts.ablDrive.parts.channelB.digitalInputs <-> AT 2/Digital inputs, state
//     PlcFastTask Inputs/GLOBAL.mtcs.parts.axes.parts.io.parts.ablDrive.parts.channelB.errorC1D <-> AT 2/Class 1 diagnostic (C1D)
//     PlcFastTask Inputs/GLOBAL.mtcs.parts.axes.parts.io.parts.ablDrive.parts.channelB.safetyOptionState <-> AT 2/Safety option state
//     PlcFastTask Inputs/GLOBAL.mtcs.parts.axes.parts.io.parts.ablDrive.parts.channelB.torqueFeedbackValue <-> AT 2/Torque feedback value
//     PlcFastTask Outputs/GLOBAL.mtcs.parts.axes.parts.io.parts.ablDrive.parts.channelA.digitalOutputs <-> MDT 1/Digital outputs
//     PlcFastTask Outputs/GLOBAL.mtcs.parts.axes.parts.io.parts.ablDrive.parts.channelA.torqueCommandValue <-> MDT 1/Torque command value
//     VISU_TASK Inputs/GLOBAL.mtcs.parts.axes.parts.io.parts.ablDrive.parts.channelA.diagnosticNumber <-> AT 1/Diagnostic number
//     VISU_TASK Inputs/GLOBAL.mtcs.parts.axes.parts.io.parts.ablDrive.parts.channelB.diagnosticNumber <-> AT 2/Diagnostic number
//   MTCS/MTCS Instance <-> ECAT (EtherCAT)/Pumps room star point - coupler (EK1101)/Pumps room star point - Slot 1 (EK1122)/REM star point (CU1128)/REM star point C (CU1128-C)/AZID (AX5206-0000-0203)
//     PlcFastTask Inputs/GLOBAL.mtcs.parts.axes.parts.io.parts.aziDrive.parts.channelA.digitalInputs <-> AT 1/Digital inputs, state
//     PlcFastTask Inputs/GLOBAL.mtcs.parts.axes.parts.io.parts.aziDrive.parts.channelA.errorC1D <-> AT 1/Class 1 diagnostic (C1D)
//     PlcFastTask Inputs/GLOBAL.mtcs.parts.axes.parts.io.parts.aziDrive.parts.channelA.safetyOptionState <-> AT 1/Safety option state
//     PlcFastTask Inputs/GLOBAL.mtcs.parts.axes.parts.io.parts.aziDrive.parts.channelA.torqueFeedbackValue <-> AT 1/Torque feedback value
//     PlcFastTask Inputs/GLOBAL.mtcs.parts.axes.parts.io.parts.aziDrive.parts.channelB.digitalInputs <-> AT 2/Digital inputs, state
//     PlcFastTask Inputs/GLOBAL.mtcs.parts.axes.parts.io.parts.aziDrive.parts.channelB.errorC1D <-> AT 2/Class 1 diagnostic (C1D)
//     PlcFastTask Inputs/GLOBAL.mtcs.parts.axes.parts.io.parts.aziDrive.parts.channelB.safetyOptionState <-> AT 2/Safety option state
//     PlcFastTask Inputs/GLOBAL.mtcs.parts.axes.parts.io.parts.aziDrive.parts.channelB.torqueFeedbackValue <-> AT 2/Torque feedback value
//     VISU_TASK Inputs/GLOBAL.mtcs.parts.axes.parts.io.parts.aziDrive.parts.channelA.diagnosticNumber <-> AT 1/Diagnostic number
//     VISU_TASK Inputs/GLOBAL.mtcs.parts.axes.parts.io.parts.aziDrive.parts.channelB.diagnosticNumber <-> AT 2/Diagnostic number
//   MTCS/MTCS Instance <-> ECAT (EtherCAT)/Pumps room star point - coupler (EK1101)/Pumps room star point - Slot 1 (EK1122)/REM star point (CU1128)/REM star point C (CU1128-C)/ELED (AX5206-0000-0203)
//     PlcFastTask Inputs/GLOBAL.mtcs.parts.axes.parts.io.parts.eleDrive.parts.channelA.digitalInputs <-> AT 1/Digital inputs, state
//     PlcFastTask Inputs/GLOBAL.mtcs.parts.axes.parts.io.parts.eleDrive.parts.channelA.errorC1D <-> AT 1/Class 1 diagnostic (C1D)
//     PlcFastTask Inputs/GLOBAL.mtcs.parts.axes.parts.io.parts.eleDrive.parts.channelA.safetyOptionState <-> AT 1/Safety option state
//     PlcFastTask Inputs/GLOBAL.mtcs.parts.axes.parts.io.parts.eleDrive.parts.channelA.torqueFeedbackValue <-> AT 1/Torque feedback value
//     PlcFastTask Inputs/GLOBAL.mtcs.parts.axes.parts.io.parts.eleDrive.parts.channelB.errorC1D <-> AT 2/Safety option state
//     PlcFastTask Outputs/GLOBAL.mtcs.parts.axes.parts.io.parts.eleDrive.parts.channelA.digitalOutputs <-> MDT 1/Digital outputs
//     VISU_TASK Inputs/GLOBAL.mtcs.parts.axes.parts.io.parts.eleDrive.parts.channelA.diagnosticNumber <-> AT 1/Diagnostic number
//     VISU_TASK Inputs/GLOBAL.mtcs.parts.axes.parts.io.parts.eleDrive.parts.channelB.diagnosticNumber <-> AT 2/Diagnostic number
//   MTCS/MTCS Instance <-> ECAT (EtherCAT)/Pumps room star point - coupler (EK1101)/Pumps room star point - Slot 1 (EK1122)/REM star point (CU1128)/REM star point C (CU1128-C)/TE:COU (EK1101)/TE:EN1 (EL5101)
//     PlcFastTask Inputs/GLOBAL.mtcs.parts.axes.parts.azi.parts.lida1._adsAddr <-> InfoData/AdsAddr
//     PlcFastTask Inputs/GLOBAL.mtcs.parts.axes.parts.azi.parts.lida1.counterValue <-> ENC Status/Counter value
//     PlcFastTask Inputs/GLOBAL.mtcs.parts.axes.parts.azi.parts.lida1.status <-> ENC Status/Status
//     PlcFastTask Outputs/GLOBAL.mtcs.parts.axes.parts.azi.parts.lida1.enableLatchC <-> ENC Control/Control/Enable latch C
//     PlcFastTask Outputs/GLOBAL.mtcs.parts.axes.parts.azi.parts.lida1.setCounter <-> ENC Control/Control/Set counter
//     PlcFastTask Outputs/GLOBAL.mtcs.parts.axes.parts.azi.parts.lida1.setCounterValue <-> ENC Control/Set counter value
//   MTCS/MTCS Instance <-> ECAT (EtherCAT)/Pumps room star point - coupler (EK1101)/Pumps room star point - Slot 1 (EK1122)/REM star point (CU1128)/REM star point C (CU1128-C)/TE:COU (EK1101)/TE:EN2 (EL5101)
//     PlcFastTask Inputs/GLOBAL.mtcs.parts.axes.parts.azi.parts.lida2._adsAddr <-> InfoData/AdsAddr
//     PlcFastTask Inputs/GLOBAL.mtcs.parts.axes.parts.azi.parts.lida2.counterValue <-> ENC Status/Counter value
//     PlcFastTask Inputs/GLOBAL.mtcs.parts.axes.parts.azi.parts.lida2.status <-> ENC Status/Status
//     PlcFastTask Outputs/GLOBAL.mtcs.parts.axes.parts.azi.parts.lida2.enableLatchC <-> ENC Control/Control/Enable latch C
//     PlcFastTask Outputs/GLOBAL.mtcs.parts.axes.parts.azi.parts.lida2.setCounter <-> ENC Control/Control/Set counter
//     PlcFastTask Outputs/GLOBAL.mtcs.parts.axes.parts.azi.parts.lida2.setCounterValue <-> ENC Control/Set counter value
//   MTCS/MTCS Instance <-> ECAT (EtherCAT)/Pumps room star point - coupler (EK1101)/Pumps room star point - Slot 1 (EK1122)/REM star point (CU1128)/REM star point C (CU1128-C)/TE:COU (EK1101)/TE:EN3 (EL5101)
//     PlcFastTask Inputs/GLOBAL.mtcs.parts.axes.parts.azi.parts.lida3._adsAddr <-> InfoData/AdsAddr
//     PlcFastTask Inputs/GLOBAL.mtcs.parts.axes.parts.azi.parts.lida3.counterValue <-> ENC Status/Counter value
//     PlcFastTask Inputs/GLOBAL.mtcs.parts.axes.parts.azi.parts.lida3.status <-> ENC Status/Status
//     PlcFastTask Outputs/GLOBAL.mtcs.parts.axes.parts.azi.parts.lida3.enableLatchC <-> ENC Control/Control/Enable latch C
//     PlcFastTask Outputs/GLOBAL.mtcs.parts.axes.parts.azi.parts.lida3.setCounter <-> ENC Control/Control/Set counter
//     PlcFastTask Outputs/GLOBAL.mtcs.parts.axes.parts.azi.parts.lida3.setCounterValue <-> ENC Control/Set counter value
//   MTCS/MTCS Instance <-> ECAT (EtherCAT)/Pumps room star point - coupler (EK1101)/Pumps room star point - Slot 1 (EK1122)/REM star point (CU1128)/REM star point C (CU1128-C)/TE:COU (EK1101)/TE:EN4 (EL5101)
//     PlcFastTask Inputs/GLOBAL.mtcs.parts.axes.parts.azi.parts.lida4._adsAddr <-> InfoData/AdsAddr
//     PlcFastTask Inputs/GLOBAL.mtcs.parts.axes.parts.azi.parts.lida4.counterValue <-> ENC Status/Counter value
//     PlcFastTask Inputs/GLOBAL.mtcs.parts.axes.parts.azi.parts.lida4.status <-> ENC Status/Status
//     PlcFastTask Outputs/GLOBAL.mtcs.parts.axes.parts.azi.parts.lida4.enableLatchC <-> ENC Control/Control/Enable latch C
//     PlcFastTask Outputs/GLOBAL.mtcs.parts.axes.parts.azi.parts.lida4.setCounter <-> ENC Control/Control/Set counter
//     PlcFastTask Outputs/GLOBAL.mtcs.parts.axes.parts.azi.parts.lida4.setCounterValue <-> ENC Control/Set counter value
//   MTCS/MTCS Instance <-> ECAT (EtherCAT)/Pumps room star point - coupler (EK1101)/Pumps room star point - Slot 1 (EK1122)/REM star point (CU1128)/REM star point C (CU1128-C)/TE:COU (EK1101)/TE:EN5 (EL5101)
//     PlcFastTask Inputs/GLOBAL.mtcs.parts.axes.parts.ele.parts.lida1._adsAddr <-> InfoData/AdsAddr
//     PlcFastTask Inputs/GLOBAL.mtcs.parts.axes.parts.ele.parts.lida1.counterValue <-> ENC Status/Counter value
//     PlcFastTask Inputs/GLOBAL.mtcs.parts.axes.parts.ele.parts.lida1.status <-> ENC Status/Status
//     PlcFastTask Outputs/GLOBAL.mtcs.parts.axes.parts.ele.parts.lida1.enableLatchC <-> ENC Control/Control/Enable latch C
//     PlcFastTask Outputs/GLOBAL.mtcs.parts.axes.parts.ele.parts.lida1.setCounter <-> ENC Control/Control/Set counter
//     PlcFastTask Outputs/GLOBAL.mtcs.parts.axes.parts.ele.parts.lida1.setCounterValue <-> ENC Control/Set counter value
//   MTCS/MTCS Instance <-> ECAT (EtherCAT)/Pumps room star point - coupler (EK1101)/Pumps room star point - Slot 1 (EK1122)/REM star point (CU1128)/REM star point C (CU1128-C)/TE:COU (EK1101)/TE:EN6 (EL5101)
//     PlcFastTask Inputs/GLOBAL.mtcs.parts.axes.parts.ele.parts.lida2._adsAddr <-> InfoData/AdsAddr
//     PlcFastTask Inputs/GLOBAL.mtcs.parts.axes.parts.ele.parts.lida2.counterValue <-> ENC Status/Counter value
//     PlcFastTask Inputs/GLOBAL.mtcs.parts.axes.parts.ele.parts.lida2.status <-> ENC Status/Status
//     PlcFastTask Outputs/GLOBAL.mtcs.parts.axes.parts.ele.parts.lida2.enableLatchC <-> ENC Control/Control/Enable latch C
//     PlcFastTask Outputs/GLOBAL.mtcs.parts.axes.parts.ele.parts.lida2.setCounter <-> ENC Control/Control/Set counter
//     PlcFastTask Outputs/GLOBAL.mtcs.parts.axes.parts.ele.parts.lida2.setCounterValue <-> ENC Control/Set counter value
//   MTCS/MTCS Instance <-> ECAT (EtherCAT)/Pumps room star point - coupler (EK1101)/Pumps room star point - Slot 1 (EK1122)/REM star point (CU1128)/REM star point C (CU1128-C)/TE:COU (EK1101)/TE:EN7 (EL5002)
//     PlcFastTask Inputs/GLOBAL.mtcs.parts.axes.parts.azi.parts.absoluteEncoder.counterValue <-> SSI Inputs Channel 1/Counter value
//     PlcFastTask Inputs/GLOBAL.mtcs.parts.axes.parts.ele.parts.absoluteEncoder.counterValue <-> SSI Inputs Channel 2/Counter value
//     VISU_TASK Inputs/GLOBAL.mtcs.parts.axes.parts.azi.parts.absoluteEncoder.status <-> SSI Inputs Channel 1/Status
//     VISU_TASK Inputs/GLOBAL.mtcs.parts.axes.parts.ele.parts.absoluteEncoder.status <-> SSI Inputs Channel 2/Status
//   MTCS/MTCS Instance <-> ECAT (EtherCAT)/Pumps room star point - coupler (EK1101)/Pumps room star point - Slot 1 (EK1122)/Timing coupler (EK1100)
//     PlcTask Inputs/GLOBAL.mtcs.parts.services.parts.timing.parts.io.parts.coupler.infoData <-> InfoData/State
//   MTCS/MTCS Instance <-> ECAT (EtherCAT)/Pumps room star point - coupler (EK1101)/Pumps room star point - Slot 1 (EK1122)/Timing coupler (EK1100)/Timing Slot 1 (serial EL6001)
//     PlcFastTask Inputs/FAST.timingSerialLine.stIn_EL6001 @bit {16..184 step 8} <-> COM Inputs/Data In {0..21}  (22 links)
//     PlcFastTask Inputs/FAST.timingSerialLine.stIn_EL6001 <-> COM Inputs/Status
//     PlcFastTask Outputs/FAST.timingSerialLine.stOut_EL6001 <-> COM Outputs/Ctrl
//     PlcFastTask Outputs/FAST.timingSerialLine.stOut_EL6001 @bit {16..184 step 8} <-> COM Outputs/Data Out {0..21}  (22 links)
//     PlcTask Inputs/GLOBAL.mtcs.parts.services.parts.timing.parts.io.parts.slot1.infoData <-> InfoData/State
//     PlcTask Inputs/GLOBAL.mtcs.parts.services.parts.timing.parts.io.parts.slot1.wcState <-> WcState/WcState
//   MTCS/MTCS Instance <-> ECAT (EtherCAT)/Pumps room star point - coupler (EK1101)/Pumps room star point - Slot 1 (EK1122)/Timing coupler (EK1100)/Timing Slot 2 (PTP EL6688)
//     PlcTask Inputs/GLOBAL.mtcs.parts.services.parts.timing.fromEL6688/externalTimestamp <-> External Sync/External time stamp
//     PlcTask Inputs/GLOBAL.mtcs.parts.services.parts.timing.fromEL6688/internalTimestamp <-> External Sync/Internal time stamp
//     PlcTask Inputs/GLOBAL.mtcs.parts.services.parts.timing.fromEL6688/notConnected <-> External Sync/External device not connected
//     PlcTask Inputs/GLOBAL.mtcs.parts.services.parts.timing.fromEL6688/updateToggle <-> External Sync/Time stamp update toggle
//     PlcTask Inputs/GLOBAL.mtcs.parts.services.parts.timing.parts.io.parts.slot2.infoData <-> InfoData/State
//     PlcTask Inputs/GLOBAL.mtcs.parts.services.parts.timing.parts.io.parts.slot2.wcState <-> WcState/WcState
//   MTCS/MTCS Instance <-> ECAT (EtherCAT)/Pumps room star point - coupler (EK1101)/Pumps room star point - Slot 2 (EK1122)/HS: Hydraulics & Safety
//     PlcTask Inputs/GLOBAL.mtcs.parts.safety.parts.io.parts.hydraulicsAndSafety.parts.COU.infoData <-> InfoData/State
//     PlcTask Inputs/GLOBAL.mtcs.parts.safety.parts.io.parts.hydraulicsAndSafety.parts.COU.wcState <-> WcState/WcState
//   MTCS/MTCS Instance <-> ECAT (EtherCAT)/Pumps room star point - coupler (EK1101)/Pumps room star point - Slot 2 (EK1122)/HS: Hydraulics & Safety/HS:AI1 (EL3102)
//     PlcTask Inputs/GLOBAL.mtcs.parts.hydraulics.parts.bottom.frequencyMeasurement.error <-> AI Standard Channel 2/Status/Error
//     PlcTask Inputs/GLOBAL.mtcs.parts.hydraulics.parts.bottom.frequencyMeasurement.overrange <-> AI Standard Channel 2/Status/Overrange
//     PlcTask Inputs/GLOBAL.mtcs.parts.hydraulics.parts.bottom.frequencyMeasurement.rawValue <-> AI Standard Channel 2/Value
//     PlcTask Inputs/GLOBAL.mtcs.parts.hydraulics.parts.bottom.frequencyMeasurement.underrange <-> AI Standard Channel 2/Status/Underrange
//     PlcTask Inputs/GLOBAL.mtcs.parts.hydraulics.parts.top.frequencyMeasurement.error <-> AI Standard Channel 1/Status/Error
//     PlcTask Inputs/GLOBAL.mtcs.parts.hydraulics.parts.top.frequencyMeasurement.overrange <-> AI Standard Channel 1/Status/Overrange
//     PlcTask Inputs/GLOBAL.mtcs.parts.hydraulics.parts.top.frequencyMeasurement.rawValue <-> AI Standard Channel 1/Value
//     PlcTask Inputs/GLOBAL.mtcs.parts.hydraulics.parts.top.frequencyMeasurement.underrange <-> AI Standard Channel 1/Status/Underrange
//     PlcTask Inputs/GLOBAL.mtcs.parts.safety.parts.io.parts.hydraulicsAndSafety.parts.AI1.infoData <-> InfoData/State
//     PlcTask Inputs/GLOBAL.mtcs.parts.safety.parts.io.parts.hydraulicsAndSafety.parts.AI1.wcState <-> WcState/WcState
//   MTCS/MTCS Instance <-> ECAT (EtherCAT)/Pumps room star point - coupler (EK1101)/Pumps room star point - Slot 2 (EK1122)/HS: Hydraulics & Safety/HS:AI2 (EL3152)
//     PlcTask Inputs/GLOBAL.mtcs.parts.hydraulics.parts.bottom.pressureMeasurement.error <-> AI Standard Channel 2/Status/Error
//     PlcTask Inputs/GLOBAL.mtcs.parts.hydraulics.parts.bottom.pressureMeasurement.overrange <-> AI Standard Channel 2/Status/Overrange
//     PlcTask Inputs/GLOBAL.mtcs.parts.hydraulics.parts.bottom.pressureMeasurement.rawValue <-> AI Standard Channel 2/Value
//     PlcTask Inputs/GLOBAL.mtcs.parts.hydraulics.parts.bottom.pressureMeasurement.underrange <-> AI Standard Channel 2/Status/Underrange
//     PlcTask Inputs/GLOBAL.mtcs.parts.hydraulics.parts.top.pressureMeasurement.error <-> AI Standard Channel 1/Status/Error
//     PlcTask Inputs/GLOBAL.mtcs.parts.hydraulics.parts.top.pressureMeasurement.overrange <-> AI Standard Channel 1/Status/Overrange
//     PlcTask Inputs/GLOBAL.mtcs.parts.hydraulics.parts.top.pressureMeasurement.rawValue <-> AI Standard Channel 1/Value
//     PlcTask Inputs/GLOBAL.mtcs.parts.hydraulics.parts.top.pressureMeasurement.underrange <-> AI Standard Channel 1/Status/Underrange
//     PlcTask Inputs/GLOBAL.mtcs.parts.safety.parts.io.parts.hydraulicsAndSafety.parts.AI2.infoData <-> InfoData/State
//     PlcTask Inputs/GLOBAL.mtcs.parts.safety.parts.io.parts.hydraulicsAndSafety.parts.AI2.wcState <-> WcState/WcState
//   MTCS/MTCS Instance <-> ECAT (EtherCAT)/Pumps room star point - coupler (EK1101)/Pumps room star point - Slot 2 (EK1122)/HS: Hydraulics & Safety/HS:AO1 (EL4132)
//     PlcTask Inputs/GLOBAL.mtcs.parts.safety.parts.io.parts.hydraulicsAndSafety.parts.AO1.infoData <-> InfoData/State
//     PlcTask Inputs/GLOBAL.mtcs.parts.safety.parts.io.parts.hydraulicsAndSafety.parts.AO1.wcState <-> WcState/WcState
//     PlcTask Outputs/GLOBAL.mtcs.parts.hydraulics.parts.bottom.driveSetpointSignal <-> Channel 2/Output
//     PlcTask Outputs/GLOBAL.mtcs.parts.hydraulics.parts.top.driveSetpointSignal <-> Channel 1/Output
//   MTCS/MTCS Instance <-> ECAT (EtherCAT)/Pumps room star point - coupler (EK1101)/Pumps room star point - Slot 2 (EK1122)/HS: Hydraulics & Safety/HS:DO1 (EL2008)
//     PlcTask Inputs/GLOBAL.mtcs.parts.safety.parts.io.parts.hydraulicsAndSafety.parts.DO1.infoData <-> InfoData/State
//     PlcTask Inputs/GLOBAL.mtcs.parts.safety.parts.io.parts.hydraulicsAndSafety.parts.DO1.wcState <-> WcState/WcState
//     PlcTask Outputs/GLOBAL.mtcs.parts.hydraulics.parts.bottom.resetDriveSignal <-> Channel 2/Output
//     PlcTask Outputs/GLOBAL.mtcs.parts.hydraulics.parts.circulationPumpRelay.digitalOutput <-> Channel 3/Output
//     PlcTask Outputs/GLOBAL.mtcs.parts.hydraulics.parts.pumpsPowerRelay.digitalOutput <-> Channel 4/Output
//     PlcTask Outputs/GLOBAL.mtcs.parts.hydraulics.parts.top.resetDriveSignal <-> Channel 1/Output
//   MTCS/MTCS Instance <-> ECAT (EtherCAT)/Pumps room star point - coupler (EK1101)/Pumps room star point - Slot 2 (EK1122)/HS: Hydraulics & Safety/HS:PWR1 (EL9410)
//     PlcTask Inputs/GLOBAL.mtcs.parts.safety.parts.io.parts.hydraulicsAndSafety.parts.PWR1.infoData <-> InfoData/State
//     PlcTask Inputs/GLOBAL.mtcs.parts.safety.parts.io.parts.hydraulicsAndSafety.parts.PWR1.wcState <-> WcState/WcState
//   MTCS/MTCS Instance <-> ECAT (EtherCAT)/Pumps room star point - coupler (EK1101)/Pumps room star point - Slot 2 (EK1122)/HS: Hydraulics & Safety/HS:RTD1 (EL3202-0010)
//     PlcTask Inputs/GLOBAL.mtcs.parts.hydraulics.bearingTemperature.error <-> RTD Inputs Channel 1/Status/Error
//     PlcTask Inputs/GLOBAL.mtcs.parts.hydraulics.bearingTemperature.overrange <-> RTD Inputs Channel 1/Status/Overrange
//     PlcTask Inputs/GLOBAL.mtcs.parts.hydraulics.bearingTemperature.rawValue <-> RTD Inputs Channel 1/Value
//     PlcTask Inputs/GLOBAL.mtcs.parts.hydraulics.bearingTemperature.underrange <-> RTD Inputs Channel 1/Status/Underrange
//     PlcTask Inputs/GLOBAL.mtcs.parts.safety.parts.io.parts.hydraulicsAndSafety.parts.RTD1.infoData <-> InfoData/State
//     PlcTask Inputs/GLOBAL.mtcs.parts.safety.parts.io.parts.hydraulicsAndSafety.parts.RTD1.wcState <-> WcState/WcState
//   MTCS/MTCS Instance <-> ECAT (EtherCAT)/Pumps room star point - coupler (EK1101)/Pumps room star point - Slot 2 (EK1122)/HS: Hydraulics & Safety/HS:SI1 (EL1904)
//     PlcTask Inputs/GLOBAL.mtcs.parts.safety.parts.hydraulics.bottomTripOK <-> Module 1 (FSOES)/TxPDO/FSOE/InputChannel2
//     PlcTask Inputs/GLOBAL.mtcs.parts.safety.parts.hydraulics.pumpsMinFrequency <-> Module 1 (FSOES)/TxPDO/FSOE/InputChannel4
//     PlcTask Inputs/GLOBAL.mtcs.parts.safety.parts.hydraulics.topTripOK <-> Module 1 (FSOES)/TxPDO/FSOE/InputChannel1
//     PlcTask Inputs/GLOBAL.mtcs.parts.safety.parts.io.parts.hydraulicsAndSafety.parts.SI1.infoData <-> InfoData/State
//     PlcTask Inputs/GLOBAL.mtcs.parts.safety.parts.io.parts.hydraulicsAndSafety.parts.SI1.wcState <-> WcState/WcState
//   MTCS/MTCS Instance <-> ECAT (EtherCAT)/Pumps room star point - coupler (EK1101)/Pumps room star point - Slot 2 (EK1122)/HS: Hydraulics & Safety/HS:SI2 (EL1904)
//     PlcTask Inputs/GLOBAL.mtcs.parts.safety.parts.io.parts.hydraulicsAndSafety.parts.SI2.infoData <-> InfoData/State
//     PlcTask Inputs/GLOBAL.mtcs.parts.safety.parts.io.parts.hydraulicsAndSafety.parts.SI2.wcState <-> WcState/WcState
//     VISU_TASK Inputs/GLOBAL.mtcs.parts.safety.parts.hydraulics.pumpsPowered <-> Module 1 (FSOES)/TxPDO/FSOE/InputChannel2
//     VISU_TASK Inputs/GLOBAL.mtcs.parts.safety.parts.hydraulics.returnFilterOverpressure <-> Module 1 (FSOES)/TxPDO/FSOE/InputChannel1
//   MTCS/MTCS Instance <-> ECAT (EtherCAT)/Pumps room star point - coupler (EK1101)/Pumps room star point - Slot 2 (EK1122)/HS: Hydraulics & Safety/HS:SI3 (EL1904)
//     PlcTask Inputs/GLOBAL.mtcs.parts.safety.parts.emergencyStops.dome1NC <-> Module 1 (FSOES)/TxPDO/FSOE/InputChannel1
//     PlcTask Inputs/GLOBAL.mtcs.parts.safety.parts.emergencyStops.dome2NC <-> Module 1 (FSOES)/TxPDO/FSOE/InputChannel2
//     PlcTask Inputs/GLOBAL.mtcs.parts.safety.parts.io.parts.hydraulicsAndSafety.parts.SI3.infoData <-> InfoData/State
//     PlcTask Inputs/GLOBAL.mtcs.parts.safety.parts.io.parts.hydraulicsAndSafety.parts.SI3.wcState <-> WcState/WcState
//     VISU_TASK Inputs/GLOBAL.mtcs.parts.safety.parts.emergencyStops.dome1NO <-> Module 1 (FSOES)/TxPDO/FSOE/InputChannel3
//     VISU_TASK Inputs/GLOBAL.mtcs.parts.safety.parts.emergencyStops.dome2NO <-> Module 1 (FSOES)/TxPDO/FSOE/InputChannel4
//   MTCS/MTCS Instance <-> ECAT (EtherCAT)/Pumps room star point - coupler (EK1101)/Pumps room star point - Slot 2 (EK1122)/HS: Hydraulics & Safety/HS:SI4 (EL1904)
//     PlcTask Inputs/GLOBAL.mtcs.parts.safety.parts.emergencyStops.controlRoomNC <-> Module 1 (FSOES)/TxPDO/FSOE/InputChannel1
//     PlcTask Inputs/GLOBAL.mtcs.parts.safety.parts.emergencyStops.firstFloorNC <-> Module 1 (FSOES)/TxPDO/FSOE/InputChannel2
//     PlcTask Inputs/GLOBAL.mtcs.parts.safety.parts.io.parts.hydraulicsAndSafety.parts.SI4.infoData <-> InfoData/State
//     PlcTask Inputs/GLOBAL.mtcs.parts.safety.parts.io.parts.hydraulicsAndSafety.parts.SI4.wcState <-> WcState/WcState
//     VISU_TASK Inputs/GLOBAL.mtcs.parts.safety.parts.emergencyStops.controlRoomNO <-> Module 1 (FSOES)/TxPDO/FSOE/InputChannel3
//     VISU_TASK Inputs/GLOBAL.mtcs.parts.safety.parts.emergencyStops.firstFloorNO <-> Module 1 (FSOES)/TxPDO/FSOE/InputChannel4
//   MTCS/MTCS Instance <-> ECAT (EtherCAT)/Pumps room star point - coupler (EK1101)/Pumps room star point - Slot 2 (EK1122)/HS: Hydraulics & Safety/HS:SL (EL6900)
//     PlcFastTask Inputs/GLOBAL.mtcs.parts.safety.parts.motionBlocking.motionAllowed <-> StandardInputs/Standard Out Var 90
//     PlcFastTask Inputs/GLOBAL.mtcs.parts.safety.parts.motionBlocking.telescopeAzimuthReleaseOK <-> StandardInputs/Standard Out Var 52
//     PlcFastTask Inputs/GLOBAL.mtcs.parts.safety.parts.motionBlocking.telescopeElevationReleaseOK <-> StandardInputs/Standard Out Var 89
//     PlcFastTask Inputs/GLOBAL.mtcs.parts.safety.parts.motionBlocking.telescopeRotationReleaseOK <-> StandardInputs/Standard Out Var 88
//     PlcFastTask Outputs/GLOBAL.mtcs.parts.axes.parts.io.parts.ablDrive.parts.channelA.safetyErrorAck <-> StandardOutputs/Standard In Var 106
//     PlcFastTask Outputs/GLOBAL.mtcs.parts.axes.parts.io.parts.ablDrive.parts.channelB.safetyErrorAck <-> StandardOutputs/Standard In Var 107
//     PlcFastTask Outputs/GLOBAL.mtcs.parts.axes.parts.io.parts.aziDrive.parts.channelA.safetyErrorAck <-> StandardOutputs/Standard In Var 104
//     PlcFastTask Outputs/GLOBAL.mtcs.parts.axes.parts.io.parts.aziDrive.parts.channelB.safetyErrorAck <-> StandardOutputs/Standard In Var 105
//     PlcFastTask Outputs/GLOBAL.mtcs.parts.axes.parts.io.parts.eleDrive.parts.channelA.safetyErrorAck <-> StandardOutputs/Standard In Var 108
//     PlcFastTask Outputs/GLOBAL.mtcs.parts.axes.parts.io.parts.eleDrive.parts.channelB.safetyErrorAck <-> StandardOutputs/Standard In Var 109
//     PlcTask Inputs/GLOBAL.mtcs.parts.safety.parts.domeAccess.groupComError <-> StandardInputs/Standard Out Var 85
//     PlcTask Inputs/GLOBAL.mtcs.parts.safety.parts.domeAccess.groupFbError <-> StandardInputs/Standard Out Var 86
//     PlcTask Inputs/GLOBAL.mtcs.parts.safety.parts.domeAccess.groupOutError <-> StandardInputs/Standard Out Var 87
//     PlcTask Inputs/GLOBAL.mtcs.parts.safety.parts.emergencyStops.allOK <-> StandardInputs/Standard Out Var 58
//     PlcTask Inputs/GLOBAL.mtcs.parts.safety.parts.emergencyStops.discrepancyError <-> StandardInputs/Standard Out Var 57
//     PlcTask Inputs/GLOBAL.mtcs.parts.safety.parts.emergencyStops.groupComError <-> StandardInputs/Standard Out Var 59
//     PlcTask Inputs/GLOBAL.mtcs.parts.safety.parts.emergencyStops.groupFbError <-> StandardInputs/Standard Out Var 61
//     PlcTask Inputs/GLOBAL.mtcs.parts.safety.parts.emergencyStops.groupOutError <-> StandardInputs/Standard Out Var 60
//     PlcTask Inputs/GLOBAL.mtcs.parts.safety.parts.hydraulics.allOK <-> StandardInputs/Standard Out Var 38
//     PlcTask Inputs/GLOBAL.mtcs.parts.safety.parts.hydraulics.groupComError <-> StandardInputs/Standard Out Var 40
//     PlcTask Inputs/GLOBAL.mtcs.parts.safety.parts.hydraulics.groupFbError <-> StandardInputs/Standard Out Var 41
//     PlcTask Inputs/GLOBAL.mtcs.parts.safety.parts.hydraulics.groupOutError <-> StandardInputs/Standard Out Var 42
//     PlcTask Inputs/GLOBAL.mtcs.parts.safety.parts.hydraulics.pressureNotRising <-> StandardInputs/Standard Out Var 66
//     PlcTask Inputs/GLOBAL.mtcs.parts.safety.parts.hydraulics.pumpsFrequencyNotRising <-> StandardInputs/Standard Out Var 65
//     PlcTask Inputs/GLOBAL.mtcs.parts.safety.parts.hydraulics.pumpsRelease <-> StandardInputs/Standard Out Var 69
//     PlcTask Inputs/GLOBAL.mtcs.parts.safety.parts.hydraulics.pumpsRunning <-> StandardInputs/Standard Out Var 72
//     PlcTask Inputs/GLOBAL.mtcs.parts.safety.parts.hydraulics.pumpsStartingUp <-> StandardInputs/Standard Out Var 70
//     PlcTask Inputs/GLOBAL.mtcs.parts.safety.parts.hydraulics.pumpsStopped <-> StandardInputs/Standard Out Var 68
//     PlcTask Inputs/GLOBAL.mtcs.parts.safety.parts.io.parts.hydraulicsAndSafety.parts.SL.infoData <-> InfoData/State
//     PlcTask Inputs/GLOBAL.mtcs.parts.safety.parts.io.parts.hydraulicsAndSafety.parts.SL.wcState <-> WcState/WcState
//     PlcTask Inputs/GLOBAL.mtcs.parts.safety.parts.motionBlocking.groupComError <-> StandardInputs/Standard Out Var 62
//     PlcTask Inputs/GLOBAL.mtcs.parts.safety.parts.motionBlocking.groupFbError <-> StandardInputs/Standard Out Var 63
//     PlcTask Inputs/GLOBAL.mtcs.parts.safety.parts.motionBlocking.groupOutError <-> StandardInputs/Standard Out Var 64
//     PlcTask Outputs/GLOBAL.mtcs.parts.safety.parts.domeAccess.errorAcknowledge <-> StandardOutputs/Standard In Var 83
//     PlcTask Outputs/GLOBAL.mtcs.parts.safety.parts.emergencyStops.errorAcknowledge <-> StandardOutputs/Standard In Var 50
//     PlcTask Outputs/GLOBAL.mtcs.parts.safety.parts.emergencyStops.restartOutput <-> StandardOutputs/Standard In Var 56
//     PlcTask Outputs/GLOBAL.mtcs.parts.safety.parts.hydraulics.errorAcknowledge <-> StandardOutputs/Standard In Var 1
//     PlcTask Outputs/GLOBAL.mtcs.parts.safety.parts.hydraulics.resetErrorsOutput <-> StandardOutputs/Standard In Var 49
//     PlcTask Outputs/GLOBAL.mtcs.parts.safety.parts.hydraulics.restartPumpsOutput <-> StandardOutputs/Standard In Var 46
//     PlcTask Outputs/GLOBAL.mtcs.parts.safety.parts.motionBlocking.errorAcknowledge <-> StandardOutputs/Standard In Var 51
//     VISU_TASK Inputs/GLOBAL.mtcs.parts.safety.parts.domeAccess.safeAccess <-> StandardInputs/Standard Out Var 103
//     VISU_TASK Inputs/GLOBAL.mtcs.parts.safety.parts.hydraulics.noOverpressure <-> StandardInputs/Standard Out Var 67
//     VISU_TASK Inputs/GLOBAL.mtcs.parts.safety.parts.hydraulics.noUnderpressure <-> StandardInputs/Standard Out Var 36
//     VISU_TASK Inputs/GLOBAL.mtcs.parts.safety.parts.hydraulics.noUnderpressureNoDelay <-> StandardInputs/Standard Out Var 35
//     VISU_TASK Inputs/GLOBAL.mtcs.parts.safety.parts.hydraulics.underpressureError <-> StandardInputs/Standard Out Var 71
//   MTCS/MTCS Instance <-> ECAT (EtherCAT)/Pumps room star point - coupler (EK1101)/Pumps room star point - Slot 2 (EK1122)/HS: Hydraulics & Safety/HS:SO1 (EL2904)
//     PlcTask Inputs/GLOBAL.mtcs.parts.safety.parts.io.parts.hydraulicsAndSafety.parts.SO1.infoData <-> InfoData/State
//     PlcTask Inputs/GLOBAL.mtcs.parts.safety.parts.io.parts.hydraulicsAndSafety.parts.SO1.wcState <-> WcState/WcState
//   MTCS/MTCS Instance <-> ECAT (EtherCAT)/Pumps room star point - coupler (EK1101)/Pumps room star point - Slot 2 (EK1122)/PG: Pumps Group
//     PlcTask Inputs/GLOBAL.mtcs.parts.hydraulics.parts.io.parts.pumpsGroup.parts.COU.infoData <-> InfoData/State
//     PlcTask Inputs/GLOBAL.mtcs.parts.hydraulics.parts.io.parts.pumpsGroup.parts.COU.wcState <-> WcState/WcState
//   MTCS/MTCS Instance <-> ECAT (EtherCAT)/Pumps room star point - coupler (EK1101)/Pumps room star point - Slot 2 (EK1122)/PG: Pumps Group/PG:DI1 (EL1008)
//     PlcTask Inputs/GLOBAL.mtcs.parts.hydraulics.circulationFilterDOK <-> Channel 2/Input
//     PlcTask Inputs/GLOBAL.mtcs.parts.hydraulics.circulationFilterGOK <-> Channel 3/Input
//     PlcTask Inputs/GLOBAL.mtcs.parts.hydraulics.oilLevelTooHigh <-> Channel 1/Input
//     PlcTask Inputs/GLOBAL.mtcs.parts.hydraulics.parts.io.parts.pumpsGroup.parts.DI1.infoData <-> InfoData/State
//     PlcTask Inputs/GLOBAL.mtcs.parts.hydraulics.parts.io.parts.pumpsGroup.parts.DI1.wcState <-> WcState/WcState
//   MTCS/MTCS Instance <-> ECAT (EtherCAT)/Pumps room star point - coupler (EK1101)/Pumps room star point - Slot 2 (EK1122)/PG: Pumps Group/PG:DI2 (EL1008)
//     PlcTask Inputs/GLOBAL.mtcs.parts.hydraulics.parts.bottom.entranceFilter{1..4}OK <-> Channel {5..8}/Input  (4 links)
//     PlcTask Inputs/GLOBAL.mtcs.parts.hydraulics.parts.io.parts.pumpsGroup.parts.DI2.infoData <-> InfoData/State
//     PlcTask Inputs/GLOBAL.mtcs.parts.hydraulics.parts.io.parts.pumpsGroup.parts.DI2.wcState <-> WcState/WcState
//     PlcTask Inputs/GLOBAL.mtcs.parts.hydraulics.parts.top.entranceFilter{1..4}OK <-> Channel {1..4}/Input  (4 links)
//   MTCS/MTCS Instance <-> ECAT (EtherCAT)/Pumps room star point - coupler (EK1101)/Pumps room star point - Slot 2 (EK1122)/PG: Pumps Group/PG:SI1 (EL1904)
//     PlcTask Inputs/GLOBAL.mtcs.parts.hydraulics.parts.io.parts.pumpsGroup.parts.SI1.infoData <-> InfoData/State
//     PlcTask Inputs/GLOBAL.mtcs.parts.hydraulics.parts.io.parts.pumpsGroup.parts.SI1.wcState <-> WcState/WcState
//     VISU_TASK Inputs/GLOBAL.mtcs.parts.safety.parts.hydraulics.bottomNoOverpressure <-> Module 1 (FSOES)/TxPDO/FSOE/InputChannel1
//     VISU_TASK Inputs/GLOBAL.mtcs.parts.safety.parts.hydraulics.topNoOverpressure <-> Module 1 (FSOES)/TxPDO/FSOE/InputChannel2
//   MTCS/MTCS Instance <-> ECAT (EtherCAT)/Pumps room star point - coupler (EK1101)/Pumps room star point - Slot 2 (EK1122)/PG: Pumps Group/PG:SI2 (EL1904)
//     PlcTask Inputs/GLOBAL.mtcs.parts.hydraulics.parts.io.parts.pumpsGroup.parts.SI2.infoData <-> InfoData/State
//     PlcTask Inputs/GLOBAL.mtcs.parts.hydraulics.parts.io.parts.pumpsGroup.parts.SI2.wcState <-> WcState/WcState
//     VISU_TASK Inputs/GLOBAL.mtcs.parts.safety.parts.hydraulics.top{1..4}NoUnderpressure <-> Module 1 (FSOES)/TxPDO/FSOE/InputChannel{1..4}  (4 links)
//   MTCS/MTCS Instance <-> ECAT (EtherCAT)/Pumps room star point - coupler (EK1101)/Pumps room star point - Slot 2 (EK1122)/PG: Pumps Group/PG:SI3 (EL1904)
//     PlcTask Inputs/GLOBAL.mtcs.parts.hydraulics.parts.io.parts.pumpsGroup.parts.SI3.infoData <-> InfoData/State
//     PlcTask Inputs/GLOBAL.mtcs.parts.hydraulics.parts.io.parts.pumpsGroup.parts.SI3.wcState <-> WcState/WcState
//     VISU_TASK Inputs/GLOBAL.mtcs.parts.safety.parts.hydraulics.bottom{5..8}NoUnderpressure <-> Module 1 (FSOES)/TxPDO/FSOE/InputChannel{1..4}  (4 links)
//   MTCS/MTCS Instance <-> ECAT (EtherCAT)/Pumps room star point - coupler (EK1101)/Pumps room star point - Slot 3 (EK1122)/DA: Dome Access
//     PlcTask Inputs/GLOBAL.mtcs.parts.safety.parts.io.parts.domeAccess.parts.COU.infoData <-> InfoData/State
//     PlcTask Inputs/GLOBAL.mtcs.parts.safety.parts.io.parts.domeAccess.parts.COU.wcState <-> WcState/WcState
//   MTCS/MTCS Instance <-> ECAT (EtherCAT)/Pumps room star point - coupler (EK1101)/Pumps room star point - Slot 3 (EK1122)/DA: Dome Access/DA:DI1 (EL1008)
//     PlcTask Inputs/GLOBAL.mtcs.parts.safety.parts.domeAccess.keypadKey{1..8} <-> Channel {1..8}/Input  (8 links)
//     PlcTask Inputs/GLOBAL.mtcs.parts.safety.parts.io.parts.domeAccess.parts.DI1.infoData <-> InfoData/State
//     PlcTask Inputs/GLOBAL.mtcs.parts.safety.parts.io.parts.domeAccess.parts.DI1.wcState <-> WcState/WcState
//   MTCS/MTCS Instance <-> ECAT (EtherCAT)/Pumps room star point - coupler (EK1101)/Pumps room star point - Slot 3 (EK1122)/DA: Dome Access/DA:DI2 (EL1008)
//     PlcTask Inputs/GLOBAL.mtcs.parts.safety.parts.domeAccess.door1Closed <-> Channel 3/Input
//     PlcTask Inputs/GLOBAL.mtcs.parts.safety.parts.domeAccess.door2Closed <-> Channel 4/Input
//     PlcTask Inputs/GLOBAL.mtcs.parts.safety.parts.domeAccess.keypadKey9 <-> Channel 1/Input
//     PlcTask Inputs/GLOBAL.mtcs.parts.safety.parts.domeAccess.keypadKeyStar <-> Channel 2/Input
//     PlcTask Inputs/GLOBAL.mtcs.parts.safety.parts.domeAccess.personHasLeftButtonPressed <-> Channel 6/Input
//     PlcTask Inputs/GLOBAL.mtcs.parts.safety.parts.domeAccess.returnButtonPressed <-> Channel 5/Input
//     PlcTask Inputs/GLOBAL.mtcs.parts.safety.parts.io.parts.domeAccess.parts.DI2.infoData <-> InfoData/State
//     PlcTask Inputs/GLOBAL.mtcs.parts.safety.parts.io.parts.domeAccess.parts.DI2.wcState <-> WcState/WcState
//   MTCS/MTCS Instance <-> ECAT (EtherCAT)/Pumps room star point - coupler (EK1101)/Pumps room star point - Slot 3 (EK1122)/DA: Dome Access/DA:DO1 (EL2008)
//     PlcFastTask Outputs/GLOBAL.mtcs.parts.safety.parts.domeAccess.personHasEntered <-> Channel 6/Output
//     PlcTask Inputs/GLOBAL.mtcs.parts.safety.parts.io.parts.domeAccess.parts.DO1.infoData <-> InfoData/State
//     PlcTask Inputs/GLOBAL.mtcs.parts.safety.parts.io.parts.domeAccess.parts.DO1.wcState <-> WcState/WcState
//     PlcTask Outputs/GLOBAL.mtcs.parts.safety.parts.domeAccess.awakeLedOn <-> Channel 3/Output
//     PlcTask Outputs/GLOBAL.mtcs.parts.safety.parts.domeAccess.buzzerSounding <-> Channel 5/Output
//     PlcTask Outputs/GLOBAL.mtcs.parts.safety.parts.domeAccess.enteredLedOn <-> Channel 1/Output
//     PlcTask Outputs/GLOBAL.mtcs.parts.safety.parts.domeAccess.movingLedOn <-> Channel 2/Output
//     PlcTask Outputs/GLOBAL.mtcs.parts.safety.parts.domeAccess.sleepingLedOn <-> Channel 4/Output
//   MTCS/MTCS Instance <-> ECAT (EtherCAT)/Pumps room star point - coupler (EK1101)/Pumps room star point - Slot 3 (EK1122)/DA: Dome Access/DA:RE1 (EL2622)
//     PlcTask Inputs/GLOBAL.mtcs.parts.safety.parts.io.parts.domeAccess.parts.RE1.infoData <-> InfoData/State
//     PlcTask Inputs/GLOBAL.mtcs.parts.safety.parts.io.parts.domeAccess.parts.RE1.wcState <-> WcState/WcState
//     PlcTask Outputs/GLOBAL.mtcs.parts.safety.parts.domeAccess.parts.lampsRelay1.digitalOutput <-> Channel 1/Output
//     PlcTask Outputs/GLOBAL.mtcs.parts.safety.parts.domeAccess.parts.lampsRelay2.digitalOutput <-> Channel 2/Output
//   MTCS/MTCS Instance <-> ECAT (EtherCAT)/Pumps room star point - coupler (EK1101)/Pumps room star point - Slot 3 (EK1122)/DA: Dome Access/DA:RE2 (EL2622)
//     PlcTask Inputs/GLOBAL.mtcs.parts.safety.parts.io.parts.domeAccess.parts.RE2.infoData <-> InfoData/State
//     PlcTask Inputs/GLOBAL.mtcs.parts.safety.parts.io.parts.domeAccess.parts.RE2.wcState <-> WcState/WcState
//     PlcTask Outputs/GLOBAL.mtcs.parts.safety.parts.domeAccess.parts.lampsRelay3.digitalOutput <-> Channel 1/Output
//     PlcTask Outputs/GLOBAL.mtcs.parts.safety.parts.domeAccess.parts.lampsRelay4.digitalOutput <-> Channel 2/Output
//   MTCS/MTCS Instance <-> ECAT (EtherCAT)/Pumps room star point - coupler (EK1101)/Pumps room star point - Slot 3 (EK1122)/DA: Dome Access/DA:SI1 (EL1904)
//     PlcTask Inputs/GLOBAL.mtcs.parts.safety.parts.emergencyStops.domeAccessNC <-> Module 1 (FSOES)/TxPDO/FSOE/InputChannel1
//     PlcTask Inputs/GLOBAL.mtcs.parts.safety.parts.io.parts.domeAccess.parts.SI1.infoData <-> InfoData/State
//     PlcTask Inputs/GLOBAL.mtcs.parts.safety.parts.io.parts.domeAccess.parts.SI1.wcState <-> WcState/WcState
//     VISU_TASK Inputs/GLOBAL.mtcs.parts.safety.parts.emergencyStops.domeAccessNO <-> Module 1 (FSOES)/TxPDO/FSOE/InputChannel2
//   MTCS/MTCS Instance <-> M3 CANopen bus/Box 1 (MCBL3006S-CO) - LINMOT
//     PlcTask Inputs/GLOBAL.mtcs.parts.m3.parts.translation.parts.motorDrive.newMilliampsValue <-> TxPDO 3/Inputs/Current Actual Value
//   MTCS/MTCS Instance <-> M3 CANopen bus/Box 2 (MCBL3006S-CO) - ROTPOS
//     PlcTask Inputs/GLOBAL.mtcs.parts.m3.parts.rotation.parts.positioningDrive.newMilliampsValue <-> TxPDO 3/Inputs/Current Actual Value
//   MTCS/MTCS Instance <-> M3 CANopen bus/Box 3 (MCBL3006S-CO) - ROTABL
//     PlcTask Inputs/GLOBAL.mtcs.parts.m3.parts.rotation.parts.antiBacklashDrive.newMilliampsValue <-> TxPDO 3/Inputs/Current Actual Value
//   MTCS/MTCS Instance <-> Fast SAF/Axes/AZI_ABL
//     PlcFastTask Inputs/GLOBAL.mtcs.parts.axes.parts.azi.parts.ablAxis.axis_ref.NcToPlc <-> Outputs/ToPlc
//     PlcFastTask Outputs/GLOBAL.mtcs.parts.axes.parts.azi.parts.ablAxis.axis_ref.PlcToNc <-> Inputs/FromPlc
//   MTCS/MTCS Instance <-> Fast SAF/Axes/AZI_Physical
//     PlcFastTask Inputs/GLOBAL.mtcs.parts.axes.parts.azi.parts.physicalAxis.axis_ref.NcToPlc <-> Outputs/ToPlc
//     PlcFastTask Outputs/GLOBAL.mtcs.parts.axes.parts.azi.parts.physicalAxis.axis_ref.PlcToNc <-> Inputs/FromPlc
//   MTCS/MTCS Instance <-> Fast SAF/Axes/AZI_Virtual
//     PlcFastTask Inputs/GLOBAL.mtcs.parts.axes.parts.azi.parts.virtualAxis.axis_ref.NcToPlc <-> Outputs/ToPlc
//     PlcFastTask Outputs/GLOBAL.mtcs.parts.axes.parts.azi.parts.virtualAxis.axis_ref.PlcToNc <-> Inputs/FromPlc
//   MTCS/MTCS Instance <-> Fast SAF/Axes/Cover_Bottom_1
//     PlcTask Inputs/GLOBAL.mtcs.parts.cover.parts.bottom.parts.p1.parts.axis.axis_ref.NcToPlc <-> Outputs/ToPlc
//     PlcTask Outputs/GLOBAL.mtcs.parts.cover.parts.bottom.parts.p1.parts.axis.axis_ref.PlcToNc <-> Inputs/FromPlc
//   MTCS/MTCS Instance <-> Fast SAF/Axes/Cover_Bottom_2
//     PlcTask Inputs/GLOBAL.mtcs.parts.cover.parts.bottom.parts.p2.parts.axis.axis_ref.NcToPlc <-> Outputs/ToPlc
//     PlcTask Outputs/GLOBAL.mtcs.parts.cover.parts.bottom.parts.p2.parts.axis.axis_ref.PlcToNc <-> Inputs/FromPlc
//   MTCS/MTCS Instance <-> Fast SAF/Axes/Cover_Bottom_3
//     PlcTask Inputs/GLOBAL.mtcs.parts.cover.parts.bottom.parts.p3.parts.axis.axis_ref.NcToPlc <-> Outputs/ToPlc
//     PlcTask Outputs/GLOBAL.mtcs.parts.cover.parts.bottom.parts.p3.parts.axis.axis_ref.PlcToNc <-> Inputs/FromPlc
//   MTCS/MTCS Instance <-> Fast SAF/Axes/Cover_Bottom_4
//     PlcTask Inputs/GLOBAL.mtcs.parts.cover.parts.bottom.parts.p4.parts.axis.axis_ref.NcToPlc <-> Outputs/ToPlc
//     PlcTask Outputs/GLOBAL.mtcs.parts.cover.parts.bottom.parts.p4.parts.axis.axis_ref.PlcToNc <-> Inputs/FromPlc
//   MTCS/MTCS Instance <-> Fast SAF/Axes/Cover_Top_1
//     PlcTask Inputs/GLOBAL.mtcs.parts.cover.parts.top.parts.p1.parts.axis.axis_ref.NcToPlc <-> Outputs/ToPlc
//     PlcTask Outputs/GLOBAL.mtcs.parts.cover.parts.top.parts.p1.parts.axis.axis_ref.PlcToNc <-> Inputs/FromPlc
//   MTCS/MTCS Instance <-> Fast SAF/Axes/Cover_Top_2
//     PlcTask Inputs/GLOBAL.mtcs.parts.cover.parts.top.parts.p2.parts.axis.axis_ref.NcToPlc <-> Outputs/ToPlc
//     PlcTask Outputs/GLOBAL.mtcs.parts.cover.parts.top.parts.p2.parts.axis.axis_ref.PlcToNc <-> Inputs/FromPlc
//   MTCS/MTCS Instance <-> Fast SAF/Axes/Cover_Top_3
//     PlcTask Inputs/GLOBAL.mtcs.parts.cover.parts.top.parts.p3.parts.axis.axis_ref.NcToPlc <-> Outputs/ToPlc
//     PlcTask Outputs/GLOBAL.mtcs.parts.cover.parts.top.parts.p3.parts.axis.axis_ref.PlcToNc <-> Inputs/FromPlc
//   MTCS/MTCS Instance <-> Fast SAF/Axes/Cover_Top_4
//     PlcTask Inputs/GLOBAL.mtcs.parts.cover.parts.top.parts.p4.parts.axis.axis_ref.NcToPlc <-> Outputs/ToPlc
//     PlcTask Outputs/GLOBAL.mtcs.parts.cover.parts.top.parts.p4.parts.axis.axis_ref.PlcToNc <-> Inputs/FromPlc
//   MTCS/MTCS Instance <-> Fast SAF/Axes/ELE_Physical
//     PlcFastTask Inputs/GLOBAL.mtcs.parts.axes.parts.ele.parts.physicalAxis.axis_ref.NcToPlc <-> Outputs/ToPlc
//     PlcFastTask Outputs/GLOBAL.mtcs.parts.axes.parts.ele.parts.physicalAxis.axis_ref.PlcToNc <-> Inputs/FromPlc
//   MTCS/MTCS Instance <-> Fast SAF/Axes/ELE_Virtual
//     PlcFastTask Inputs/GLOBAL.mtcs.parts.axes.parts.ele.parts.virtualAxis.axis_ref.NcToPlc <-> Outputs/ToPlc
//     PlcFastTask Outputs/GLOBAL.mtcs.parts.axes.parts.ele.parts.virtualAxis.axis_ref.PlcToNc <-> Inputs/FromPlc
//   MTCS/MTCS Instance <-> Fast SAF/Axes/M3_RotationAntiBacklash
//     PlcTask Inputs/GLOBAL.mtcs.parts.m3.parts.rotation.parts.antiBacklashAxis.axis_ref.NcToPlc <-> Outputs/ToPlc
//     PlcTask Outputs/GLOBAL.mtcs.parts.m3.parts.rotation.parts.antiBacklashAxis.axis_ref.PlcToNc <-> Inputs/FromPlc
//   MTCS/MTCS Instance <-> Fast SAF/Axes/M3_RotationPosHall
//     PlcTask Inputs/GLOBAL.mtcs.parts.m3.parts.rotation.parts.positioningHallAxis.axis_ref.NcToPlc <-> Outputs/ToPlc
//     PlcTask Outputs/GLOBAL.mtcs.parts.m3.parts.rotation.parts.positioningHallAxis.axis_ref.PlcToNc <-> Inputs/FromPlc
//   MTCS/MTCS Instance <-> Fast SAF/Axes/M3_RotationPositioning
//     PlcTask Inputs/GLOBAL.mtcs.parts.m3.parts.rotation.parts.positioningAxis.axis_ref.NcToPlc <-> Outputs/ToPlc
//     PlcTask Outputs/GLOBAL.mtcs.parts.m3.parts.rotation.parts.positioningAxis.axis_ref.PlcToNc <-> Inputs/FromPlc
//   MTCS/MTCS Instance <-> Fast SAF/Axes/M3_Translation
//     PlcTask Inputs/GLOBAL.mtcs.parts.m3.parts.translation.parts.motorAxis.axis_ref.NcToPlc <-> Outputs/ToPlc
//     PlcTask Outputs/GLOBAL.mtcs.parts.m3.parts.translation.parts.motorAxis.axis_ref.PlcToNc <-> Inputs/FromPlc
//   MTCS/MTCS Instance <-> Fast SAF/Axes/ROC_Physical
//     PlcFastTask Inputs/GLOBAL.mtcs.parts.axes.parts.roc.parts.physicalAxis.axis_ref.NcToPlc <-> Outputs/ToPlc
//     PlcFastTask Outputs/GLOBAL.mtcs.parts.axes.parts.roc.parts.physicalAxis.axis_ref.PlcToNc <-> Inputs/FromPlc
//   MTCS/MTCS Instance <-> Fast SAF/Axes/ROC_Virtual
//     PlcFastTask Inputs/GLOBAL.mtcs.parts.axes.parts.roc.parts.virtualAxis.axis_ref.NcToPlc <-> Outputs/ToPlc
//     PlcFastTask Outputs/GLOBAL.mtcs.parts.axes.parts.roc.parts.virtualAxis.axis_ref.PlcToNc <-> Inputs/FromPlc
//   MTCS/MTCS Instance <-> Fast SAF/Axes/RON_Physical
//     PlcFastTask Inputs/GLOBAL.mtcs.parts.axes.parts.ron.parts.physicalAxis.axis_ref.NcToPlc <-> Outputs/ToPlc
//     PlcFastTask Outputs/GLOBAL.mtcs.parts.axes.parts.ron.parts.physicalAxis.axis_ref.PlcToNc <-> Inputs/FromPlc
//   MTCS/MTCS Instance <-> Fast SAF/Axes/RON_Virtual
//     PlcFastTask Inputs/GLOBAL.mtcs.parts.axes.parts.ron.parts.virtualAxis.axis_ref.NcToPlc <-> Outputs/ToPlc
//     PlcFastTask Outputs/GLOBAL.mtcs.parts.axes.parts.ron.parts.virtualAxis.axis_ref.PlcToNc <-> Inputs/FromPlc
//   MTCS/MTCS Instance <-> Slalib/TelescopePointing
//     PlcFastTask Inputs/GLOBAL.mtcs.parts.axes.fromCppAxes <-> Outputs/toPlc/toAxes
//     PlcFastTask Inputs/GLOBAL.mtcs.parts.services.parts.timing.fromCppTiming <-> Outputs/toPlc/toTiming
//     PlcFastTask Outputs/GLOBAL.mtcs.parts.axes.toCppAxes <-> Inputs/fromPlc/fromAxes
//     PlcTask Outputs/GLOBAL.mtcs.parts.services.parts.timing.toCppTiming <-> Inputs/fromPlc/fromTiming

CONFIGURATION MTCS
    RESOURCE PLC ON TwinCAT3
        TASK PlcFastTask(INTERVAL := T#2ms, PRIORITY := 8);
        TASK PlcTask(INTERVAL := T#10ms, PRIORITY := 14);
        TASK VISU_TASK(INTERVAL := T#100000us, PRIORITY := 16);
        PROGRAM FAST WITH PlcFastTask : FAST;
        PROGRAM MAIN WITH PlcTask : MAIN;
        PROGRAM VisuElems_Visu_Prg WITH VISU_TASK : VisuElems.Visu_Prg;
    END_RESOURCE
END_CONFIGURATION

// ---- MTCS/Axes/Helper/AxesFastTaskAxisIO.TcDUT
TYPE AxesFastTaskAxisIO :
STRUCT
	virtual_fromNc    AT %I* : NCTOPLC_AXIS_REF;
	physical_fromPlc  AT %I* : PLCTONC_AXIS_REF;
	physical_toNc     AT %Q* : PLCTONC_AXIS_REF;
END_STRUCT
END_TYPE

// ---- MTCS/Axes/Helper/HoursMinutesSeconds.TcDUT
TYPE HoursMinutesSeconds :
STRUCT
    positive : BOOL;
    
    hours : DINT;
    minutes : DINT;
    seconds : LREAL;
END_STRUCT
END_TYPE

// ---- MTCS/Axes/Helper/DegreesMinutesSeconds.TcDUT
TYPE DegreesMinutesSeconds :
STRUCT
    positive : BOOL;
    
    degrees : DINT;
    minutes : DINT;
    seconds : LREAL;
END_STRUCT
END_TYPE

// ---- MTCS/Axes/Widgets/AxesDialogRotUnits.TcDUT
TYPE AxesDialogRotUnits :
(
	DIALOG_DMS := 0,
    DIALOG_DEGREES := 1,
    DIALOG_RADIANS := 2
);
END_TYPE

// ---- MTCS/Axes/Widgets/AxesRotationAxisTabs.TcDUT
TYPE AxesRotationAxisTabs :
(
	OVERVIEW := 0,
    PROCESSES := 1,
    DRIVE_CHANNEL := 2,
    VIRTUAL_AXIS := 3,
    PHYSICAL_AXIS := 4
);
END_TYPE

// ---- MTCS/Axes/Widgets/AxesManualTabs.TcDUT
TYPE AxesManualTabs :
(
	TAB_POSITIONS := 0,
    TAB_JOYSTICK_AZIELE := 1,
    TAB_JOYSTICK_ROT := 2,
    TAB_OFFSETS_AZIELE := 3,
    TAB_OFFSETS_ALPHADELTA := 4,
    TAB_MOVEABSOLUTE := 5,
    TAB_MOVEVELOCITY  := 6
);
END_TYPE

// ---- MTCS/Axes/Widgets/AxesElevationAxisTabs.TcDUT
TYPE AxesElevationAxisTabs :
(
	OVERVIEW := 0,
    PROCESSES := 1,
    DRIVE_CHANNEL := 2,
    VIRTUAL_AXIS := 3,
    PHYSICAL_AXIS := 4,
    LIDAS := 5,
    ABSOLUTE_ENCODER := 6
);
END_TYPE

// ---- MTCS/Axes/Widgets/AxesAzimuthAxisTabs.TcDUT
TYPE AxesAzimuthAxisTabs :
(
	OVERVIEW := 0,
    PROCESSES := 1,
    AZI_DRIVE_CHANNEL := 2,
    ABL_DRIVE_CHANNEL := 3,
    VIRTUAL_AXIS := 4,
    PHYSICAL_AXIS := 5,
    ABL_AXIS  := 6,
    LIDAS := 7,
    ABSOLUTE_ENCODER := 8
);
END_TYPE

// ---- MTCS/Axes/Widgets/AxesDialogSign.TcDUT
TYPE AxesDialogSign :
(
	DIALOG_PLUS := 0,
    DIALOG_MINUS := 1
);
END_TYPE

// ---- MTCS/Axes/Widgets/AxesAxesTabs.TcDUT
TYPE AxesAxesTabs :
(
	AZI := 0,
    ELE := 2,
    ROC := 3,
    RON := 4,
    FW  := 5
);
END_TYPE

// ---- MTCS/Axes/Widgets/AxesMoveProcessWidgetUnits.TcDUT
TYPE AxesMoveProcessWidgetUnits :
(
	DEGMINSEC := 0,
    DEGREES := 1,
    ARCMINUTES := 2,
    ARCSECCONDS := 3,
    RADIANS := 4
);
END_TYPE

// ---- MTCS/Axes/Widgets/AxesDialogAlphaUnits.TcDUT
TYPE AxesDialogAlphaUnits :
(
	DIALOG_HMS := 0,
    DIALOG_HOURS := 1,
    DIALOG_RADIANS := 2
);
END_TYPE

// ---- MTCS/Axes/Widgets/AxesDialogDeltaUnits.TcDUT
TYPE AxesDialogDeltaUnits :
(
	DIALOG_DMS := 0,
    DIALOG_DEGREES := 1,
    DIALOG_RADIANS := 2
);
END_TYPE

// ---- MTCS/Axes/Widgets/AxesTabs.TcDUT
TYPE AxesTabs :
(
	OVERVIEW := 0,
	MANUAL := 1,
    AXES := 2,
	TARGET := 3,
    TPOINT := 4,
    ADVANCED := 5,
    IO := 6,
    CONFIG := 7
);
END_TYPE

// ---- MTCS/Common/HelperCode/StatusColor.TcDUT
TYPE StatusColor :
STRUCT
    fg : Colors; // foreground
    bg : Colors; // background
END_STRUCT
END_TYPE

// ---- MTCS/Common/Widgets/Colors.TcDUT
TYPE Colors :
(
	GREEN := 16#FF00FF00,
	RED := 16#FFFF0000,
	ORANGE := 16#FFFF802D,
	GRAY := 16#FFD3D3D3,
	DARK_GRAY := 16#FF949494,
	BLACK := 16#FF000000,
	WHITE := 16#FFFFFFFF,
	BLUE := 16#FF0000FF
) DWORD;
END_TYPE

// ---- MTCS/Cover/Widgets/CoverConfigTabs.TcDUT
TYPE CoverConfigTabs :
(
	GENERAL := 0,
    TOP := 1,
    BOTTOM := 2,
    TOP_1 := 3,
    TOP_2 := 4,
    TOP_3 := 5,
    TOP_4 := 6,
    BOTTOM_1 := 7,
    BOTTOM_2 := 8,
    BOTTOM_3 := 9,
    BOTTOM_4 := 10
);
END_TYPE

// ---- MTCS/Cover/Widgets/CoverTabs.TcDUT
TYPE CoverTabs :
(
	OVERVIEW := 0,
    TOP := 1,
    BOTTOM := 2,
    IO := 3,
    CONFIG := 4
);
END_TYPE

// ---- MTCS/Hydraulics/Widgets/HydraulicsTabs.TcDUT
TYPE HydraulicsTabs :
(
	OVERVIEW := 0,
    TECHNICAL := 1,
    IO := 2,
    CONFIG := 3
);
END_TYPE

// ---- MTCS/M1/Widgets/M1Tabs.TcDUT
TYPE M1Tabs :
(
	OVERVIEW := 0,
    RADIAL := 1,
    AXIAL := 2,
    IO := 3,
    CONFIG := 4
);
END_TYPE

// ---- MTCS/MTCS/MtcsGlobalConfig.TcDUT
TYPE MtcsGlobalConfig :
STRUCT

    SIMULATION_ACTIVE               : BOOL := FALSE;
    
    PASSWORD_TECH : STRING := '1512'; // birth year of Gerardus Mercator :)
    
    STARTUP_WAIT_TIME : TIME := T#3S;
    
    PLC_TASK_TIME : TIME := T#10MS;
    PLC_CTRL_TIME : TIME := T#10MS;
    PLC_FAST_TASK_TIME : TIME := T#2MS;
    SLALIB_TASK_TIME : TIME := T#10MS;
	PLC_TASK_FLIP : BOOL; // constantly flips (True -> False -> True -> ...)
    
    
    PLC_FAST_TASK_START_MS          : LREAL;
    PLC_FAST_TASK_PREVIOUS_START_MS : LREAL;
    PLC_FAST_MEASURED_TASK_TIME_MS  : LREAL;
    
    SYSTEM_TIME : GETSYSTEMTIME; // the actual system time
    TIME_NOW_MS : LREAL;         // the actual time in milliseconds
    TIME_NOW_S : LREAL;         // the actual time in seconds
    
    MTCS_EDITABLE_CONFIG_SYMBOL_NAME   : STRING := 'GLOBAL.mtcs.editableConfig';
    MTCS_ACTIVE_CONFIG_SYMBOL_NAME     : STRING := 'GLOBAL.mtcs.config';
    MTCS_CONFIG_FILE_PATH              : STRING := 'C:\MTCS_Config\Mtcs.xml';
    
    AXES_EDITABLE_CONFIG_SYMBOL_NAME   : STRING := 'GLOBAL.mtcs.parts.axes.editableConfig';
    AXES_ACTIVE_CONFIG_SYMBOL_NAME     : STRING := 'GLOBAL.mtcs.parts.axes.config';
    AXES_CONFIG_FILE_PATH              : STRING := 'C:\MTCS_Config\Axes.xml';
    
    COVER_EDITABLE_CONFIG_SYMBOL_NAME   : STRING := 'GLOBAL.mtcs.parts.cover.editableConfig';
    COVER_ACTIVE_CONFIG_SYMBOL_NAME     : STRING := 'GLOBAL.mtcs.parts.cover.config';
    COVER_CONFIG_FILE_PATH              : STRING := 'C:\MTCS_Config\Cover.xml';
    
    M1_EDITABLE_CONFIG_SYMBOL_NAME   : STRING := 'GLOBAL.mtcs.parts.m1.editableConfig';
    M1_ACTIVE_CONFIG_SYMBOL_NAME     : STRING := 'GLOBAL.mtcs.parts.m1.config';
    M1_CONFIG_FILE_PATH              : STRING := 'C:\MTCS_Config\M1.xml';
    
    M2_EDITABLE_CONFIG_SYMBOL_NAME   : STRING := 'GLOBAL.mtcs.parts.m2.editableConfig';
    M2_ACTIVE_CONFIG_SYMBOL_NAME     : STRING := 'GLOBAL.mtcs.parts.m2.config';
    M2_CONFIG_FILE_PATH              : STRING := 'C:\MTCS_Config\M2.xml';
    
    M3_EDITABLE_CONFIG_SYMBOL_NAME   : STRING := 'GLOBAL.mtcs.parts.m3.editableConfig';
    M3_ACTIVE_CONFIG_SYMBOL_NAME     : STRING := 'GLOBAL.mtcs.parts.m3.config';
    M3_CONFIG_FILE_PATH              : STRING := 'C:\MTCS_Config\M3.xml';
    
    SERVICES_EDITABLE_CONFIG_SYMBOL_NAME   : STRING := 'GLOBAL.mtcs.parts.services.editableConfig';
    SERVICES_ACTIVE_CONFIG_SYMBOL_NAME     : STRING := 'GLOBAL.mtcs.parts.services.config';
    SERVICES_CONFIG_FILE_PATH              : STRING := 'C:\MTCS_Config\Services.xml';
    
    TElEMETRY_EDITABLE_CONFIG_SYMBOL_NAME   : STRING := 'GLOBAL.mtcs.parts.telemetry.editableConfig';
    TElEMETRY_ACTIVE_CONFIG_SYMBOL_NAME     : STRING := 'GLOBAL.mtcs.parts.telemetry.config';
    TElEMETRY_CONFIG_FILE_PATH              : STRING := 'C:\MTCS_Config\Telemetry.xml';
    
    HYDRAULICS_EDITABLE_CONFIG_SYMBOL_NAME   : STRING := 'GLOBAL.mtcs.parts.hydraulics.editableConfig';
    HYDRAULICS_ACTIVE_CONFIG_SYMBOL_NAME     : STRING := 'GLOBAL.mtcs.parts.hydraulics.config';
    HYDRAULICS_CONFIG_FILE_PATH              : STRING := 'C:\MTCS_Config\Hydraulics.xml';
    
    SAFETY_EDITABLE_CONFIG_SYMBOL_NAME   : STRING := 'GLOBAL.mtcs.parts.safety.editableConfig';
    SAFETY_ACTIVE_CONFIG_SYMBOL_NAME     : STRING := 'GLOBAL.mtcs.parts.safety.config';
    SAFETY_CONFIG_FILE_PATH              : STRING := 'C:\MTCS_Config\Safety.xml';
    
    AXES_TPOINT_EDITABLE_CONFIG_SYMBOL_PREFIX : STRING :=  'GLOBAL.mtcs.parts.axes.parts.tpoint.parts.'; // + 'model?' + SUFFIX
    AXES_TPOINT_EDITABLE_CONFIG_SYMBOL_SUFFIX : STRING :=  '.editableConfig'; 
    AXES_TPOINT_ACTIVE_CONFIG_SYMBOL_PREFIX   : STRING :=  'GLOBAL.mtcs.parts.axes.parts.tpoint.parts.'; // + 'model?' + SUFFIX
    AXES_TPOINT_ACTIVE_CONFIG_SYMBOL_SUFFIX   : STRING :=  '.config'; 
    AXES_TPOINT_CONFIG_FILE_PATH_PREFIX       : STRING := 'C:\MTCS_Config\TPoint\'; // + 'instrument?' + SUFFIX
    AXES_TPOINT_CONFIG_FILE_PATH_SUFFIX       : STRING := '.xml';
    
END_STRUCT
END_TYPE

// ---- GVLs/GLOBAL.TcGVL
VAR_GLOBAL
    
    // declare the global config FIRST (so it is initialized before all the rest *)
    config : MTCSGlobalConfig;
    
	mtcs : MTCS;
    
	{attribute 'OPC.UA.DA' := '0'}
	gui : MTCSWidget;
    
    
END_VAR

// ---- GVLs/REMANENT.TcGVL
VAR_GLOBAL
END_VAR

(* below are some "special" variables wich must be stored persistently in memory. *)
(* !!! NOTE !!!
   New declarations only can be added at the end of the list. 
   At a download those will be detected as "new" and will not demand a 
   re-initialization of the complete list. *)

VAR_GLOBAL RETAIN PERSISTENT
    
    (* The following variables represent the actual values
       of the Faulhaber drives of the rotation mechanism of M3.
       They are continuously updated, so at all times they correspond to the
       actual value. When the PLC software starts, these
       values will be written back to the axes. If the axes have not
       moved, then they will be again (more or less) at the same position,
       just like an absolute encoder. It' s not very precise, but it' s good
       enough in 99% of the cases because M3 is positioned using an absolute
       encoder. The "semi-absolute" motor position values are only needed to 
       maintain a certain offset between both motors, in order to apply a
       counter-acting torque by the magnetic clutch. This doesn' t have to
       be very accurate, hence we can use the approach of storing them
       in the persistent memory of the PLC. 
       In case these values get lost, a new calibration procedure is needed. *)
	M3_ROTPOS_POSITION: LREAL; // positioning motor of the rotation mechanism
    M3_ROTABL_POSITION: LREAL; // anti-backlash motor of the rotation mechanism
END_VAR

// ---- POUs/FAST.TcPOU
PROGRAM FAST
VAR
    startTimer : TON;
    
    
    timingSerialLine : SerialLine;
    m2FastTaskControl : M2FastTaskControl;
	
	tempSafetyState : INT;
	tempSafetyTon : TON;
	restartEStop AT %Q* : BOOL;
	safetyGroupAck AT %Q* : BOOL;
	EStopError AT %I* : BOOL;
	EnableDrive AT %I* : BOOL;
	outputEnableDrive AT %Q* : BOOL;
	
END_VAR

startTimer(IN := TRUE, PT := GLOBAL.config.STARTUP_WAIT_TIME + T#1s); // wait one second longer, because the FAST task depends on the normal PLC task!

// update the actual times
GLOBAL.config.SYSTEM_TIME();
GLOBAL.config.TIME_NOW_MS := (UDINT_TO_LREAL(GLOBAL.config.SYSTEM_TIME.timeHiDW)*429496.7296) + (UDINT_TO_LREAL(GLOBAL.config.SYSTEM_TIME.timeLoDW)/10000);
GLOBAL.config.TIME_NOW_S := GLOBAL.config.TIME_NOW_MS / 1000.0;

GLOBAL.config.PLC_FAST_TASK_PREVIOUS_START_MS   := GLOBAL.config.PLC_FAST_TASK_START_MS;
GLOBAL.config.PLC_FAST_TASK_START_MS            := GLOBAL.config.TIME_NOW_MS;
GLOBAL.config.PLC_FAST_MEASURED_TASK_TIME_MS    := GLOBAL.config.PLC_FAST_TASK_START_MS - GLOBAL.config.PLC_FAST_TASK_PREVIOUS_START_MS;



IF startTimer.Q THEN
    
    timingSerialLine(
            TxBuffer := GLOBAL.mtcs.parts.services.parts.timing.parts.serialInfo.TxBuffer,
            RxBuffer := GLOBAL.mtcs.parts.services.parts.timing.parts.serialInfo.RxBuffer);
    
    m2FastTaskControl(
            brakeReleaseSignal := GLOBAL.mtcs.parts.m2.parts.multiplexer.parts.release.digitalOutput,
            actualCounterValue := GLOBAL.mtcs.parts.m2.parts.moveStepsProcedure.actualCounterValue);
    
    // the whole axes subsystem runs within the FAST task!
    GLOBAL.mtcs.parts.axes(
        timing := GLOBAL.mtcs.parts.services.parts.timing,
        motionBlocking := GLOBAL.mtcs.parts.safety.parts.motionBlocking,
        domeAccess := GLOBAL.mtcs.parts.safety.parts.domeAccess,
        operatorStatus := GLOBAL.mtcs.statuses.operatorStatus,
        activityStatus := GLOBAL.mtcs.statuses.activityStatus,
        activeInstrument := GLOBAL.mtcs.activeInstrument,
        isInstrumentActive := GLOBAL.mtcs.isInstrumentActive);
    

END_IF

END_PROGRAM

// ---- MTCS/Common/HelperCode/SerialLine.TcPOU
FUNCTION_BLOCK SerialLine
VAR_INPUT
    stIn_EL6001  AT %I* : EL6inData22B;
    stOut_EL6001 AT %Q* : EL6outData22B;
END_VAR
VAR_OUTPUT
    Error   : BOOL;
    ErrorID : INT;
    ErrorDescription : STRING;
END_VAR
VAR_IN_OUT
   TxBuffer : ComBuffer;
   RxBuffer : ComBuffer;
END_VAR
VAR
    control : SerialLineControl;
END_VAR

control(
    Mode      := ComSerialLineMode_t.SERIALLINEMODE_EL6_22B,
    pComIn    := ADR(stIn_EL6001),
    pComOut   := ADR(stOut_EL6001),
    SizeComIn := SIZEOF(stIn_EL6001),
    TxBuffer  := TxBuffer,
    RxBuffer  := RxBuffer,
    Error     => Error,
    ErrorID   => ErrorID);

ErrorDescription := ComErrorToString(control.ErrorID);

END_FUNCTION_BLOCK

// ---- MTCS/Common/HelperCode/ComErrorToString.TcPOU
FUNCTION ComErrorToString : STRING
VAR_INPUT
    errorId : ComError_t;
END_VAR
VAR
END_VAR

CASE ErrorID OF
    ComError_t.COMERROR_NOERROR:                ComErrorToString := 'No error';
    ComError_t.COMERROR_PARAMETERCHANGED:       ComErrorToString := 'Parameter changed';
    ComError_t.COMERROR_TXBUFFOVERRUN:          ComErrorToString := 'Tx buffer overrun';
    ComError_t.COMERROR_STRINGOVERRUN:          ComErrorToString := 'String overrun';
    ComError_t.COMERROR_ZEROCHARINVALID:        ComErrorToString := 'Zero char invalid';
    ComError_t.COMERROR_INVALIDPOINTER:         ComErrorToString := 'Invalid pointer';
    ComError_t.COMERROR_INVALIDRXPOINTER:       ComErrorToString := 'Invalid Rx pointer';
    ComError_t.COMERROR_INVALIDRXLENGTH:        ComErrorToString := 'Invalid Rx length';
    ComError_t.COMERROR_DATASIZEOVERRUN:        ComErrorToString := 'Datasize overrun';
    ComError_t.COMERROR_INVALIDPROCESSDATASIZE: ComErrorToString := 'Invalid process data size';
    ComError_t.COMERROR_MODENOTSUPPORTED:       ComErrorToString := 'Mode not supported';
    ComError_t.COMERROR_INVALIDCHANNELNUMBER:   ComErrorToString := 'Invalid channel number';
    ComError_t.COMERROR_INVALIDBAUDRATE:        ComErrorToString := 'Invalid baudrate';
    ComError_t.COMERROR_INVALIDNUMDATABITS:     ComErrorToString := 'Invalid number of data bits';
    ComError_t.COMERROR_INVALIDNUMSTOPBITS:     ComErrorToString := 'Invalid number of stop bits';
    ComError_t.COMERROR_INVALIDPARITY:          ComErrorToString := 'Invalid parity';
    ComError_t.COMERROR_INVALIDHANDSHAKE:       ComErrorToString := 'Invalid handshake';
    ComError_t.COMERROR_INVALIDNUMREGISTERS:    ComErrorToString := 'Invalid number of registers';
    ComError_t.COMERROR_INVALIDREGISTER:        ComErrorToString := 'Invalid register';
    ComError_t.COMERROR_TIMEOUT:                ComErrorToString := 'Timeout';
END_CASE

END_FUNCTION

// ---- MTCS/MTCS/StateMachines/MTCS.TcPOU
FUNCTION_BLOCK MTCS EXTENDS SM_MTCS
VAR_INPUT
END_VAR
VAR_OUTPUT
END_VAR
VAR
    _initializingCurrentAction : INT;
    _onFirstStartCurrentAction : INT;
	
	_nt_reboot : NT_Reboot;
	_nt_shutdown : NT_Shutdown;
    
    _wakeUpState : INT;
    _goToSleepState : INT;
    _changeInstrumentState : INT;
    _changeInstrumentConfig : InstrumentConfig;
END_VAR

// flip the PLC_TASK_FLIP bool once every cycle
GLOBAL.config.PLC_TASK_FLIP := NOT GLOBAL.config.PLC_TASK_FLIP;

_update();

_onFirstStart();
_locking();
_initializing();
_changingOperator();
_verifyingPassword();
_locking();
_unlocking();
_rebooting();
_shuttingDown();
_wakingUp();
_goingToSleep();
_changingInstrument();

_update();

METHOD _onFirstStart
VAR_INPUT
END_VAR
CASE _onFirstStartCurrentAction OF
    0:
        // start loading the config from XML file
        parts.configManager.processes.load.start(parts.configManager.processes.load.set.filePath);
        _onFirstStartCurrentAction := 1;
    1:
        // wait until the config has been loaded
        IF parts.configManager.processes.load.statuses.busyStatus.idle THEN
            IF parts.configManager.processes.load.statuses.healthStatus.good THEN
                _onFirstStartCurrentAction := 2;
            ELSE
                _onFirstStartCurrentAction := 999;
            END_IF
        END_IF
    2:
        // now start activating the config
        parts.configManager.processes.activate.start();
        _onFirstStartCurrentAction := 3;
    3:
        // wait until the config has been activated
        IF parts.configManager.processes.activate.statuses.busyStatus.idle THEN
            IF parts.configManager.processes.activate.statuses.healthStatus.good THEN
                _onFirstStartCurrentAction := 4;
            ELSE
                _onFirstStartCurrentAction := 999;
            END_IF
        END_IF
    4:
        // nothing to do, done!
        ;
    999:
        // error, but nothing we can do about it now!
        ;

END_CASE
END_METHOD

METHOD _update
VAR_INPUT
END_VAR
SUPER^();


IF  (parts.axes.statuses.initializationStatus.initialized OR parts.axes.statuses.initializationStatus.locked) AND 
    (parts.cover.statuses.initializationStatus.initialized OR parts.cover.statuses.initializationStatus.locked) AND 
    (parts.hydraulics.statuses.initializationStatus.initialized OR parts.hydraulics.statuses.initializationStatus.locked) AND 
    (parts.m1.statuses.initializationStatus.initialized OR parts.m1.statuses.initializationStatus.locked) AND 
    (parts.m2.statuses.initializationStatus.initialized OR parts.m2.statuses.initializationStatus.locked) AND 
    (parts.m3.statuses.initializationStatus.initialized OR parts.m3.statuses.initializationStatus.locked) AND 
    (parts.safety.statuses.initializationStatus.initialized OR parts.safety.statuses.initializationStatus.locked) AND 
    (parts.services.statuses.initializationStatus.initialized OR parts.services.statuses.initializationStatus.locked) AND 
    (parts.telemetry.statuses.initializationStatus.initialized OR parts.telemetry.statuses.initializationStatus.locked) THEN
    
            statuses.initializationStatus(superState := TRUE, state := InitializationStates.INITIALIZED);
            
ELSIF  parts.axes.statuses.initializationStatus.initializingFailed OR 
    parts.cover.statuses.initializationStatus.initializingFailed OR 
    parts.hydraulics.statuses.initializationStatus.initializingFailed OR 
    parts.m1.statuses.initializationStatus.initializingFailed OR 
    parts.m2.statuses.initializationStatus.initializingFailed OR 
    parts.m3.statuses.initializationStatus.initializingFailed OR 
    parts.safety.statuses.initializationStatus.initializingFailed OR 
    parts.services.statuses.initializationStatus.initializingFailed OR 
    parts.telemetry.statuses.initializationStatus.initializingFailed THEN
    
            statuses.initializationStatus(superState := TRUE, state := InitializationStates.INITIALIZING_FAILED);
            
ELSIF  parts.axes.statuses.initializationStatus.initializing OR 
    parts.cover.statuses.initializationStatus.initializing OR 
    parts.hydraulics.statuses.initializationStatus.initializing OR 
    parts.m1.statuses.initializationStatus.initializing OR 
    parts.m2.statuses.initializationStatus.initializing OR 
    parts.m3.statuses.initializationStatus.initializing OR 
    parts.safety.statuses.initializationStatus.initializing OR 
    parts.services.statuses.initializationStatus.initializing OR 
    parts.telemetry.statuses.initializationStatus.initializing THEN
    
            statuses.initializationStatus(superState := TRUE, state := InitializationStates.INITIALIZING);
            
